// TwinCAT 3 PLC project ExternControl
// ProgramVersion: 3.1.4026.22
// libraries:
//   Tc2_Standard, * (Beckhoff Automation GmbH)
//   Tc2_System, * (Beckhoff Automation GmbH)
//   Tc2_Utilities, * (Beckhoff Automation GmbH)
// project tree:
//   CAM/types/ ST_CAM_CTRL.TcDUT, ST_CAM_DATA.TcDUT (not stored), ST_CAM_INFO.TcDUT (not stored), ST_CAM_OPTIONS.TcDUT (not stored), ST_CAM_READ_VALUES_PARAMETER.TcDUT, ST_CAM_SCALING_DATA.TcDUT, ST_CAM_STATE.TcDUT (not stored), ST_MOTION_FUNCTION.TcDUT, ST_MOTION_FUNCTION_POINT.TcDUT (not stored)
//   FLYING_SAW/ GVL_FLYING_SAW.TcGVL
//   FLYING_SAW/types/ ST_FLY_CTRL.TcDUT (not stored), ST_FLY_DATA.TcDUT (not stored), ST_FLY_OPTIONS.TcDUT (not stored), ST_FLY_STATE.TcDUT (not stored), ST_FLY_SYNC_MODE.TcDUT (not stored)
//   FUNCTIONS/TOUCH_PROBE/types/ ST_2BIT.TcDUT (not stored), ST_CTRL_TOUCH_PROBE.TcDUT, ST_DC_Input.TcDUT, ST_MTI_INPUT.TcDUT, ST_MTI_STATUS.TcDUT, ST_STATE_TOUCH_PROBE.TcDUT
//   FUNCTIONS/TRIGGER_BOX/types/ ST_CTRL_TRIGGER.TcDUT, ST_DC_Output.TcDUT (not stored), ST_DC_State.TcDUT (not stored), ST_STATE_TRIGGER.TcDUT (not stored), T_TriggerControlBits.TcDUT (not stored)
//   / GlobalTextList.TcGTLO (not stored), MAIN.TcPOU, PlcTask.TcTTO, Visualization Manager.TcVMO (not stored)
//   MAPPING/ MAPPING_out.TcPOU, MAPPING_in.TcPOU
//   MAPPING/types/ U_AXIS_CTRL.TcDUT (not stored), U_AXIS_GEAR_IN.TcDUT (not stored), U_AXIS_HOMING.TcDUT (not stored), U_AXIS_INFO.TcDUT (not stored), U_AXIS_MOTION_OPTIONS.TcDUT, U_AXIS_MOVE_DATA.TcDUT (not stored), U_AXIS_NC_PARAMETER_RD.TcDUT, U_AXIS_NC_PARAMETER_WRT.TcDUT (not stored), U_AXIS_STATE.TcDUT (not stored), U_CAM_CTRL.TcDUT (not stored), U_CAM_DATA.TcDUT (not stored), U_CAM_INFO.TcDUT, U_CAM_STATE.TcDUT (not stored), U_FLY_CTRL.TcDUT, U_FLY_DATA.TcDUT, U_FLY_OPTIONS.TcDUT, U_FLY_STATE.TcDUT, U_NCI_AXIS_ID_GROUP.TcDUT (not stored), U_NCI_CTRL.TcDUT (not stored), U_NCI_INDEX_GROUP.TcDUT, U_NCI_R_PARAMETER_I.TcDUT, U_NCI_R_PARAMETER_Q.TcDUT, U_NCI_STATE.TcDUT, U_TOUCH_PROBE_CTRL.TcDUT, U_TOUCH_PROBE_STATE.TcDUT (not stored), U_TRIGGER_CTRL.TcDUT, U_TRIGGER_STATE.TcDUT (not stored)
//   NCI/types/ E_NCI_CHANNEL_ERROR.TcDUT (not stored), E_NCI_CTRL.TcDUT (not stored), E_NCI_INTERPRETER_STATE.TcDUT, E_NCI_STATE.TcDUT (not stored), ST_3D_Group.TcDUT, ST_Index_Group.TcDUT (not stored), ST_Interface_Group.TcDUT (not stored), ST_NciChannel_Ref.TcDUT, ST_NCI_CTRL.TcDUT, ST_NCI_M_FUNC.TcDUT, ST_NCI_STATE.TcDUT (not stored), ST_R_Parameter.TcDUT
//   NC_PTP/types/axis/ E_AxisEncoderType.TcDUT, ST_HomeParams.TcDUT (not stored), ST_HomingOptionsExt.TcDUT
//   NC_PTP/types/control/ E_AXIS_CTRL.TcDUT (not stored), E_AXIS_STATE.TcDUT (not stored), ST_AXIS_CTRL.TcDUT, ST_AXIS_INFO.TcDUT (not stored), ST_AXIS_STATE.TcDUT (not stored), ST_GEAR_IN.TcDUT, ST_HOMING.TcDUT (not stored), ST_MOTION_OPTIONS.TcDUT (not stored), ST_MOVE_DATA.TcDUT, ST_NC_PARAMETER.TcDUT (not stored)
//   TEST_MOTION/ TEST.TcPOU
//   _DUT/ f_GetProgress.TcPOU, f_GetState.TcPOU, E_CHECK_STATE.TcDUT, E_PROGRESS.TcDUT
//   _GVL/ GVL_AXIS.TcGVL, GVL_CAM.TcGVL (not stored), GVL_FUNCTIONS.TcGVL (not stored), GVL_MSG.TcGVL, PLC_CONSTANT.TcGVL
//   _MSG/ fb_LocalTime.TcPOU, fb_MessageData.TcPOU, fb_MessageDataCtrl.TcPOU, f_MessageSet.TcPOU, I_MessageData.TcIO
//   _MSG/types/ e_Device.TcDUT, E_MessageType.TcDUT, E_MESSAGE_BATCH.TcDUT, E_MESSAGE_CHECK.TcDUT, E_MESSAGE_CTRL.TcDUT, E_MESSAGE_FLOW.TcDUT, E_MESSAGE_STATE.TcDUT, e_Subdevice.TcDUT, ST_Message.TcDUT, ST_MESSAGE_CTRL.TcDUT, ST_MESSAGE_STATE.TcDUT, TL_E_MESSAGETYPE.TcTLO
// real-time tasks:
//   TASK PlcTask: cycle T#1ms, priority 20, ADS port 350
//   TASK PlcTask1: cycle T#1ms, priority 1, ADS port 351
// motion (NC):
//   TASK NC-Task 1 SAF: cycle T#2ms, priority 4, ADS port 501
//   TASK NC-Task 1 SVB: cycle T#10ms, priority 8, ADS port 511
//   AXIS Axis 1 (id 1)
//     OtherSettings: AllowMotionCmdToSlave=true
//     encoder EncType=1
//     drive DrvType=5
//       Analog: TorqueSetpointScale=10, ScaleFactorActTorque=0.1
//       TimeComp: TaskDelayCycles=1
//     controller CtrType=1
//       CtrPara: PriorControlFactor=1
//         Observer: BandWidth=20
//   AXIS Axis 2 (id 2)
//     OtherSettings: AllowMotionCmdToSlave=true
//     encoder EncType=1
//     drive DrvType=5
//       Analog: TorqueSetpointScale=10, ScaleFactorActTorque=0.1
//       TimeComp: TaskDelayCycles=1
//     controller CtrType=1
//       CtrPara: PriorControlFactor=1
//         Observer: BandWidth=20
//   AXIS Axis 3 (id 3)
//     OtherSettings: AllowMotionCmdToSlave=true
//     encoder EncType=1
//     drive DrvType=5
//       Analog: TorqueSetpointScale=10, ScaleFactorActTorque=0.1
//       TimeComp: TaskDelayCycles=1
//     controller CtrType=1
//       CtrPara: PriorControlFactor=1
//         Observer: BandWidth=20
//   AXIS Axis 4 (id 4)
//     OtherSettings: AllowMotionCmdToSlave=true
//     encoder EncType=1
//     drive DrvType=5
//       Analog: TorqueSetpointScale=10, ScaleFactorActTorque=0.1
//       TimeComp: TaskDelayCycles=1
//     controller CtrType=1
//       CtrPara: PriorControlFactor=1
//         Observer: BandWidth=20
//   AXIS Axis 5 (id 5)
//     OtherSettings: AllowMotionCmdToSlave=true
//     encoder EncType=1
//     drive DrvType=5
//       Analog: TorqueSetpointScale=10, ScaleFactorActTorque=0.1
//       TimeComp: TaskDelayCycles=1
//     controller CtrType=1
//       CtrPara: PriorControlFactor=1
//         Observer: BandWidth=20
//   AXIS Axis 6 (id 6)
//     OtherSettings: AllowMotionCmdToSlave=true
//     encoder EncType=1
//     drive DrvType=5
//       Analog: TorqueSetpointScale=10, ScaleFactorActTorque=0.1
//       TimeComp: TaskDelayCycles=1
//     controller CtrType=1
//       CtrPara: PriorControlFactor=1
//         Observer: BandWidth=20
// variable links:
//   ExternControl/ExternControl Instance <-> PLC_MOTION/PLC_MOTION Instance
//     PlcTask Inputs/MAIN.eInitPlcMotion <-> PlcTask Outputs/MAIN_AXIS.eInit
//     PlcTask Inputs/MAPPING_in.AxisInfo.byState <-> PlcTask Outputs/MAPPING_AXIS_out.AxisInfo.byState
//     PlcTask Inputs/MAPPING_in.AxisParameterRd.byState <-> PlcTask Outputs/MAPPING_AXIS_out.AxisParameterOut.byState
//     PlcTask Inputs/MAPPING_in.AxisState.byState <-> PlcTask Outputs/MAPPING_AXIS_out.AxisState.byState
//     PlcTask Inputs/MAPPING_in.FlyState.byState <-> PlcTask Outputs/MAPPING_AXIS_out.FlyState.byState
//     PlcTask Outputs/MAPPING_out.AxisCtrl.byCtrl <-> PlcTask Inputs/MAPPING_AXIS_in.AxisCtrl.byCtrl
//     PlcTask Outputs/MAPPING_out.AxisGearInData.byCtrl <-> PlcTask Inputs/MAPPING_AXIS_in.AxisGearInData.byCtrl
//     PlcTask Outputs/MAPPING_out.AxisHoming.byCtrl <-> PlcTask Inputs/MAPPING_AXIS_in.AxisHoming.byCtrl
//     PlcTask Outputs/MAPPING_out.AxisMotionOptions.byCtrl <-> PlcTask Inputs/MAPPING_AXIS_in.AxisMotionOptions.byCtrl
//     PlcTask Outputs/MAPPING_out.AxisMoveData.byCtrl <-> PlcTask Inputs/MAPPING_AXIS_in.AxisMoveData.byCtrl
//     PlcTask Outputs/MAPPING_out.AxisParameterWrt.byCtrl <-> PlcTask Inputs/MAPPING_AXIS_in.AxisParameterIn.byCtrl
//     PlcTask Outputs/MAPPING_out.FlyControl.byCtrl <-> PlcTask Inputs/MAPPING_AXIS_in.FlyControl.byCtrl
//     PlcTask Outputs/MAPPING_out.FlyData.byCtrl <-> PlcTask Inputs/MAPPING_AXIS_in.FlyData.byCtrl
//     PlcTask Outputs/MAPPING_out.FlyOptions.byCtrl <-> PlcTask Inputs/MAPPING_AXIS_in.FlyOptions.byCtrl
//   PLC_MOTION/PLC_MOTION Instance <-> NC-Task 1 SAF/Axes/Axis 1
//     PlcTask Inputs/GVL_AXIS.AxisRef[1].NcToPlc <-> Outputs/ToPlc
//     PlcTask Outputs/GVL_AXIS.AxisRef[1].PlcToNc <-> Inputs/FromPlc
//   PLC_MOTION/PLC_MOTION Instance <-> NC-Task 1 SAF/Axes/Axis 2
//     PlcTask Inputs/GVL_AXIS.AxisRef[2].NcToPlc <-> Outputs/ToPlc
//     PlcTask Outputs/GVL_AXIS.AxisRef[2].PlcToNc <-> Inputs/FromPlc
//   PLC_MOTION/PLC_MOTION Instance <-> NC-Task 1 SAF/Axes/Axis 3
//     PlcTask Inputs/GVL_AXIS.AxisRef[3].NcToPlc <-> Outputs/ToPlc
//     PlcTask Outputs/GVL_AXIS.AxisRef[3].PlcToNc <-> Inputs/FromPlc
//   PLC_MOTION/PLC_MOTION Instance <-> NC-Task 1 SAF/Axes/Axis 4
//     PlcTask Inputs/GVL_AXIS.AxisRef[4].NcToPlc <-> Outputs/ToPlc
//     PlcTask Outputs/GVL_AXIS.AxisRef[4].PlcToNc <-> Inputs/FromPlc
//   PLC_MOTION/PLC_MOTION Instance <-> NC-Task 1 SAF/Axes/Axis 5
//     PlcTask Inputs/GVL_AXIS.AxisRef[5].NcToPlc <-> Outputs/ToPlc
//     PlcTask Outputs/GVL_AXIS.AxisRef[5].PlcToNc <-> Inputs/FromPlc
//   PLC_MOTION/PLC_MOTION Instance <-> NC-Task 1 SAF/Axes/Axis 6
//     PlcTask Inputs/GVL_AXIS.AxisRef[6].NcToPlc <-> Outputs/ToPlc
//     PlcTask Outputs/GVL_AXIS.AxisRef[6].PlcToNc <-> Inputs/FromPlc

CONFIGURATION ExternControl
    RESOURCE PLC ON TwinCAT3
        TASK PlcTask(INTERVAL := T#1ms, PRIORITY := 20);
        PROGRAM MAPPING_in WITH PlcTask : MAPPING_in;
        PROGRAM MAIN WITH PlcTask : MAIN;
        PROGRAM MAPPING_out WITH PlcTask : MAPPING_out;
    END_RESOURCE
END_CONFIGURATION

// ---- CAM/types/ST_CAM_CTRL.TcDUT
{attribute 'pack_mode' := '2'}
TYPE ST_CAM_CTRL :
STRUCT
  eCmd               : E_AXIS_CTRL;    // commanded axis function
END_STRUCT
END_TYPE

// ---- CAM/types/ST_CAM_READ_VALUES_PARAMETER.TcDUT
{attribute 'pack_mode' := '2'}
TYPE ST_CAM_READ_VALUES_PARAMETER :
STRUCT
  nValueSelectMask        : UINT;   // ReadMotionFunctionValues
  rValueMasterStart       : LREAL;  // ReadMotionFunctionValues
  rValueMasterEnd         : LREAL;  // ReadMotionFunctionValues
  rIncrement              : LREAL;
END_STRUCT
END_TYPE

// ---- CAM/types/ST_CAM_SCALING_DATA.TcDUT
{attribute 'pack_mode' := '2'}
TYPE ST_CAM_SCALING_DATA :
STRUCT
  bMasterRelative         : BIT;
  bSlaveRelative          : BIT;

  // scaling of X-axis (Master) of the CAM
  nMasterScalingMode      : UINT;
  rMasterOffset           : LREAL;
  rMasterScaling          : LREAL := 1.0;

  // scaling of Y-axis (Slave) of CAM
  nSlaveScalingMode       : UINT;

  rSlaveOffset            : LREAL;
  rSlaveScaling           : LREAL := 1.0;
END_STRUCT
END_TYPE

// ---- CAM/types/ST_MOTION_FUNCTION.TcDUT
{attribute 'pack_mode' := '2'}
TYPE ST_MOTION_FUNCTION :
STRUCT
  stMotionFunction            : ARRAY[1..MAX_MOTION_FUNCTION_POINTS] OF ST_MOTION_FUNCTION_POINT;
  nMotionFunctionSize         : UINT;
  nPoints                     : UINT; // number of points used in motion function 
END_STRUCT
END_TYPE

// ---- FUNCTIONS/TOUCH_PROBE/types/ST_CTRL_TOUCH_PROBE.TcDUT
TYPE ST_CTRL_TOUCH_PROBE :
STRUCT
  Enable        : BIT;

  AxisId        : UDINT;      // TwinCAT NC Axis ID

  SensorIndex   : UDINT;      // sensor select; 1 := upper , 2 := lower, 0 := default upper 

  Direction     : INT := 1;   // typeof(MC_DIRECTION)
                                // MC_Positive_Direction := 1,   -(set trigger when crossing moving in pos dir)
                                // MC_Shortest_Way,               (not used in TouchProbe or TriggerBox)
                                // MC_Negative_Direction := 3,   -(set trigger when crossing moving in neg dir)
                                // MC_Current_Direction  := 4,    (not used in TouchProbe or TriggerBox)
                                // MC_Undefined_Direction := 128  (not used in TouchProbe or TriggerBox)

  PositionStart : LREAL; // axis has to reach this position in order to start the check for change in input timestamp
  PositionEnd   : LREAL; // axis must not reach this position without state change on input --> error
END_STRUCT
END_TYPE

// ---- FUNCTIONS/TOUCH_PROBE/types/ST_DC_Input.TcDUT
TYPE ST_DC_Input :
STRUCT
  Input      : BIT;

  Status     : USINT;

  LatchPositive  : ULINT;
  LatchNegative  : ULINT;
END_STRUCT
END_TYPE

// ---- FUNCTIONS/TOUCH_PROBE/types/ST_MTI_INPUT.TcDUT
TYPE ST_MTI_INPUT :
STRUCT
  EventState            : BIT;
  EventTime             : UDINT;
END_STRUCT
END_TYPE

// ---- FUNCTIONS/TOUCH_PROBE/types/ST_MTI_STATUS.TcDUT
TYPE ST_MTI_STATUS :
STRUCT
  EventCount            : USINT;
  InputState            : BIT;
  InputBufferOverflow   : BIT;
  InputCycleCounter     : ST_2BIT;
  CountsInBuffer        : USINT;
  InputOrderFeedback    : usint;
END_STRUCT
END_TYPE

// ---- FUNCTIONS/TOUCH_PROBE/types/ST_STATE_TOUCH_PROBE.TcDUT
TYPE ST_STATE_TOUCH_PROBE :
STRUCT
  State           : UINT;   // 0 := deactivated, 100 := BUSY, 1000 := DONE, 9000 := ERROR
  LatchPositive   : LREAL;  // rising edge
  LatchNegative   : LREAL;  // falling edge
END_STRUCT
END_TYPE

// ---- FUNCTIONS/TRIGGER_BOX/types/ST_CTRL_TRIGGER.TcDUT
TYPE ST_CTRL_TRIGGER :
STRUCT
  Control             : T_TriggerControlBits;

   {attribute 'hide'}
  byc : ARRAY[1..7] OF BYTE;;


  AxisId              : UDINT;  // TwinCAT NC Axis ID

  TriggerCount        : UDINT;  // how many TriggerPositions shall be used

  TriggerPosition     : ARRAY[1..MAX_TRIGGER_COUNT] OF LREAL;  // Axis Position where output must be set by TriggerBox
                                // Trigger is set when crossing Position
END_STRUCT
END_TYPE

// ---- MAPPING/types/U_AXIS_MOTION_OPTIONS.TcDUT
TYPE U_AXIS_MOTION_OPTIONS :
UNION

  stCtrl              : ARRAY[1..MAX_AXIS] OF ST_MOTION_OPTIONS;

  byCtrl    AT %Q*    : ARRAY[1..MAX_AXIS] OF
                        ARRAY[1..SIZEOF(ST_MOTION_OPTIONS)] OF BYTE;
END_UNION
END_TYPE

// ---- MAPPING/types/U_AXIS_NC_PARAMETER_RD.TcDUT
TYPE U_AXIS_NC_PARAMETER_RD :
UNION

  stState             : ARRAY[1..MAX_AXIS] OF ST_NC_PARAMETER;

  byState   AT %I*    : ARRAY[1..MAX_AXIS] OF
                        ARRAY[1..SIZEOF(ST_NC_PARAMETER)] OF BYTE;
END_UNION
END_TYPE

// ---- MAPPING/types/U_CAM_INFO.TcDUT
TYPE U_CAM_INFO :
UNION

  stState             : ARRAY[1..MAX_AXIS] OF ST_CAM_INFO;

  byState  AT %i*     : ARRAY[1..MAX_AXIS] OF
                        ARRAY[1..SIZEOF(ST_CAM_INFO)] OF BYTE;
END_UNION
END_TYPE

// ---- MAPPING/types/U_FLY_CTRL.TcDUT
TYPE U_FLY_CTRL :
UNION

  stCtrl              : ARRAY[1..MAX_AXIS] OF ST_FLY_CTRL;

  byCtrl    AT %Q*    : ARRAY[1..MAX_AXIS] OF
                        ARRAY[1..SIZEOF(ST_FLY_CTRL)] OF BYTE;

END_UNION
END_TYPE

// ---- MAPPING/types/U_FLY_DATA.TcDUT
TYPE U_FLY_DATA :
UNION

  stCtrl              : ARRAY[1..MAX_AXIS] OF ST_FLY_DATA;

  byCtrl    AT %Q*    : ARRAY[1..MAX_AXIS] OF
                        ARRAY[1..SIZEOF(ST_FLY_DATA)] OF BYTE;

END_UNION
END_TYPE

// ---- MAPPING/types/U_FLY_OPTIONS.TcDUT
TYPE U_FLY_OPTIONS :
UNION

  stCtrl              : ARRAY[1..MAX_AXIS] OF ST_FLY_OPTIONS;

  byCtrl    AT %Q*    : ARRAY[1..MAX_AXIS] OF
                        ARRAY[1..SIZEOF(ST_FLY_OPTIONS)] OF BYTE;

END_UNION
END_TYPE

// ---- MAPPING/types/U_FLY_STATE.TcDUT
TYPE U_FLY_STATE :
UNION

  stState             : ARRAY[1..MAX_AXIS] OF ST_FLY_STATE;

  byState   AT %I*    : ARRAY[1..MAX_AXIS] OF
                        ARRAY[1..SIZEOF(ST_FLY_STATE)] OF BYTE;
END_UNION
END_TYPE

// ---- MAPPING/types/U_NCI_INDEX_GROUP.TcDUT
TYPE U_NCI_INDEX_GROUP :
UNION

  stCtrl              : ARRAY[1..MAX_NCI_CH] OF ST_Index_Group;

  byCtrl    AT %q*    : ARRAY[1..MAX_NCI_CH] OF
                        ARRAY[1..SIZEOF(ST_Index_Group)] OF BYTE;
END_UNION
END_TYPE

// ---- MAPPING/types/U_NCI_R_PARAMETER_I.TcDUT
TYPE U_NCI_R_PARAMETER_I :
UNION

  stCtrl              : ARRAY[1..MAX_NCI_CH] OF ST_R_Parameter;

  byCtrl    AT %q*    : ARRAY[1..MAX_NCI_CH] OF
                        ARRAY[1..SIZEOF(ST_R_Parameter)] OF BYTE;
END_UNION
END_TYPE

// ---- MAPPING/types/U_NCI_R_PARAMETER_Q.TcDUT
TYPE U_NCI_R_PARAMETER_Q :
UNION

  stCtrl              : ARRAY[1..MAX_NCI_CH] OF ST_R_Parameter;

  byCtrl    AT %i*    : ARRAY[1..MAX_NCI_CH] OF
                        ARRAY[1..SIZEOF(ST_R_Parameter)] OF BYTE;
END_UNION
END_TYPE

// ---- MAPPING/types/U_NCI_STATE.TcDUT
TYPE U_NCI_STATE :
UNION

  stState             : ARRAY[1..MAX_NCI_CH] OF ST_NCI_STATE;

  byState   AT %i*    : ARRAY[1..MAX_NCI_CH] OF
                        ARRAY[1..SIZEOF(ST_NCI_STATE)] OF BYTE;
END_UNION
END_TYPE

// ---- MAPPING/types/U_TOUCH_PROBE_CTRL.TcDUT
TYPE U_TOUCH_PROBE_CTRL :
UNION
  stCtrl              : ARRAY[1..MAX_TOUCH_PROBE] OF ST_CTRL_TOUCH_PROBE;

  byCtrl    AT %q*    : ARRAY[1..MAX_TOUCH_PROBE] OF
                        ARRAY[1..SIZEOF(ST_CTRL_TOUCH_PROBE)] OF BYTE;
END_UNION
END_TYPE

// ---- MAPPING/types/U_TRIGGER_CTRL.TcDUT
TYPE U_TRIGGER_CTRL :
UNION
  stCtrl              : ARRAY[1..MAX_TRIGGER_BOX] OF ST_CTRL_TRIGGER;

  byCtrl    AT %q*    : ARRAY[1..MAX_TRIGGER_BOX] OF
                        ARRAY[1..SIZEOF(ST_CTRL_TRIGGER)] OF BYTE;
END_UNION
END_TYPE

// ---- NCI/types/E_NCI_INTERPRETER_STATE.TcDUT
// Interpreter state, see also library tc2_nci.Global_Variables.NCI_INTERPRETER_xxx
//  Date    Name  Version   Remarks
//  2016/09/29  FJK   1.0     1st Version
{attribute -'to_string'}
TYPE E_NCI_INTERPRETER_STATE :
(
  NCI_INTERPRETER_INITFAILED := 0,
  NCI_INTERPRETER_IDLE := 1,
  NCI_INTERPRETER_READY := 2,
  NCI_INTERPRETER_STARTED := 3,
  NCI_INTERPRETER_SCANNING := 4,
  NCI_INTERPRETER_RUNNING := 5,
  NCI_INTERPRETER_STAY_RUNNING := 6,
  NCI_INTERPRETER_WRITETABLE := 7,
  NCI_INTERPRETER_SEARCHLINE := 8,
  NCI_INTERPRETER_END := 9,
  NCI_INTERPRETER_SINGLESTOP := 10, 
  NCI_INTERPRETER_ABORTING := 11,
  NCI_INTERPRETER_ABORTED := 12,
  NCI_INTERPRETER_FAULT := 13,
  NCI_INTERPRETER_RESET := 14,
  NCI_INTERPRETER_STOP := 15,
  NCI_INTERPRETER_WAITFUNC := 16,
  NCI_INTERPRETER_FLUSHBUFFERS := 17
) DWORD;    //Basis-Datentyp
END_TYPE

// ---- NCI/types/ST_3D_Group.TcDUT
{attribute 'pack_mode' := '2'}
TYPE ST_3D_Group :
STRUCT
  nXAxisId    : UDINT := 1;
  nYAxisId    : UDINT := 2;
  nZAxisId    : UDINT := 3;
  nQ1AxisId   : UDINT;
  nQ2AxisId   : UDINT;
  nQ3AxisId   : UDINT;
  nQ4AxisId   : UDINT;
  nQ5AxisId   : UDINT;
END_STRUCT
END_TYPE

// ---- NCI/types/ST_NciChannel_Ref.TcDUT
TYPE ST_NciChannel_Ref :
STRUCT
  NcToPlc AT %I*: NcToPlc_NciChannel_Ref;   //  Externer Datentyp!
  PlcToNc AT %Q*: PlcToNc_NciChannel_Ref;   //  Externer Datentyp!
END_STRUCT
END_TYPE

// ---- NCI/types/ST_NCI_CTRL.TcDUT
{attribute 'pack_mode' := '2'}
TYPE ST_NCI_CTRL :
STRUCT
  eCmd          : E_NCI_CTRL := E_NCI_CTRL.INIT;
  rOverride     : REAL := 47.11;

  sProgramName  : STRING(255);
END_STRUCT
END_TYPE

// ---- NCI/types/ST_NCI_M_FUNC.TcDUT
{attribute 'pack_mode' := '2'}
TYPE ST_NCI_M_FUNC :
STRUCT
  FastMFuncMask   : ARRAY [1..5] OF DWORD;
  HskMFuncNo      : UINT;
  HskMFuncReq     : WORD;
  HFuncValue      : UDINT; 

  MFuncGranted    : UINT;
END_STRUCT
END_TYPE

// ---- NCI/types/ST_R_Parameter.TcDUT
{attribute 'pack_mode' := '2'}
TYPE ST_R_Parameter :
STRUCT
  _nStart               : DINT := 901;
  _nCount               : DINT :=   4;
  _rValue               : ARRAY[0..MAX_R_PARA] OF LREAL;
END_STRUCT
END_TYPE

// ---- NC_PTP/types/axis/E_AxisEncoderType.TcDUT
{attribute 'to_string'}
TYPE E_AxisEncoderType :
(
  NoEncoder := 0,
  
  Simulation_Encoder,
  
  M3000_Enc,
  M31x0_M2000_Enc,
  MDP_511_Enc,
  MDP_500_501_Enc,
  MDP_510_Enc,
  KL30xx_Enc,
  SERCOS_EtherCAT_SoE_Pos,
  SERCOS_EtherCAT_SoE_Pos_Velo,
  Binary_Enc,
  M2510_Enc,
  FOX50_Enc                     := 12,
  AX2000_Lightbus               := 14,
  Provi_DriveMC_Simodrive_611U,
  Universal_Encoder_varBitmask,
  NC_Backplane,
  spec_CANopen_Typ,
  MDP_513_DS402,
  AX2xx_B900,
  KL5151_Encoder                := 21,
  IP5209_Encoder                := 24,
  KL2531_KL2541_Encoder,
  KL2532_KL2542_Encoder,
  Time_Base_Encoder,
  TCom_Encoder_SoftDrive
)UDINT;
END_TYPE

// ---- NC_PTP/types/axis/ST_HomingOptionsExt.TcDUT
TYPE ST_HomingOptionsExt :
STRUCT
  // in order for extern control to be 
  // fully independent of any library types
  // struct is built with base types
  ClearPositionLag      : BOOL;
  SearchDirection       : INT;    // MC_Direction
  SearchVelocity        : LREAL;
  SyncDirection         : INT;    // MC_Direction
  SyncVelocity          : LREAL;
  ReferenceMode         : UDINT;  // E_EncoderReferenceMode
END_STRUCT
END_TYPE

// ---- NC_PTP/types/control/ST_AXIS_CTRL.TcDUT
{attribute 'pack_mode' := '2'}
TYPE ST_AXIS_CTRL :
STRUCT
  eCmd                : E_AXIS_CTRL;    // commanded axis function
  eProgress           : E_PROGRESS;     // progress command for synced functions
END_STRUCT
END_TYPE

// ---- NC_PTP/types/control/ST_GEAR_IN.TcDUT
{attribute 'pack_mode' := '2'}
TYPE ST_GEAR_IN :
STRUCT
  bAdvancedSlaveDynamics  : BOOL;
  nMultiMasterSyncMode    : INT;

  nAxisIndexMaster    : ARRAY [1..4] OF BYTE; // Index of Master1-4
  rGearRatio          : ARRAY [1..4] OF REAL; 
  Acceleration        : REAL;
  Deceleration        : REAL;
  Jerk                : REAL;  
END_STRUCT
END_TYPE

// ---- NC_PTP/types/control/ST_MOVE_DATA.TcDUT
{attribute 'pack_mode' := '2'}
TYPE ST_MOVE_DATA :
STRUCT
  rSetPos           : LREAL;
  rSetVelo          : LREAL;
  rOverride         : LREAL := 100.0;
  rAcc              : LREAL;
  rDec              : LREAL;
  rJerk             : LREAL;
  iDirection        : INT;
END_STRUCT
END_TYPE

// ---- _DUT/E_CHECK_STATE.TcDUT
{attribute 'qualified_only'}
{attribute 'strict'}
{attribute 'to_string'}
TYPE E_CHECK_STATE :
(
  CHECK_INIT,
  AXIS_INDEX_OUT_OF_RANGE         :=  10,

	AXIS_REF_POINTER_INVALID        := 100,
  AXIS_CTRL_POINTER_INVALID,
  AXIS_STATE_POINTER_INVALID,
  AXIS_INFO_POINTER_INVALID,
  AXIS_DATA_POINTER_INVALID,
  AXIS_NC_PARAMETER_POINTER_INVALID,
  AXIS_HOME_PARAMETER_POINTER_INVALID,
  AXIS_GEAR_IN_PARAMETER_POINTER_INVALID,
  AXIS_GEAR_IN_MULTIMASTER_POINTER_INVALID,
  AXIS_MOTION_OPTIONS_POINTER_INVALID,

  NCI_NOT_ACTIVATED               := 200,
  NCI_CHANNEL_REF_POINTER_INVALID,
  NCI_AXIS_CONFIG_POINTER_INVALID,
  NCI_MCS_AXIS_POINTER_INVALID,
  NCI_AUX_AXIS_POINTER_INVALID,
  NCI_CTRL_POINTER_INVALID,
  NCI_STATE_POINTER_INVALID,
  NCI_R_PARAMETER_READ_POINTER_INVALID,
  NCI_R_PARAMETER_wRITE_POINTER_INVALID,
  NCI_M_FUNC_POINTER_INVALID,

  CAM_NOT_ACTIVATED               := 300,
  CAM_SLAVE_AXIS_REF_INVALID,
  CAM_SLAVE_ITF_MC_AXIS_INVALID,
  CAM_MASTER_AXIS_REF_INVALID,
  CAM_MOTION_FUNCTION_POINTER_INVALID,
  CAM_MOTION_FUNCTION_POINT_POINTER_INVALID,

  CHECK_DONE                      := 10000
  
)UINT;
END_TYPE

// ---- _DUT/E_PROGRESS.TcDUT
{attribute 'qualified_only'}
//{attribute 'strict'}
{attribute 'to_string'}
TYPE E_PROGRESS :
(
  // progress has 2 use cases
  // 1. as offset to cyclic interface's state 
  //    for the requested command/function
  //    e.g. State := <Enum equivalent to eCmd> + E_PROGRESS
  //
  // 2. as state feedback (result) from (any) method
  PROGRESS_INVALID,
  PROGRESS_NOT_EXIST      :=   100,
  PROGRESS_INIT           :=  1000,
  PROGRESS_BUSY           :=  2000,
  PROGRESS_PREPARE        :=  3000,
  PROGRESS_STARTUP        :=  4000,
  PROGRESS_CHECK          :=  5000,
  PROGRESS_OCCUPIED       :=  6000,
  PROGRESS_WORKING        :=  7000,
  PROGRESS_STILL_WORKING  :=  8000,
  PROGRESS_ERROR          :=  9000,
  PROGRESS_DONE           := 10000
)UINT;
END_TYPE

// ---- _MSG/types/e_Device.TcDUT
{attribute 'to_string'}
TYPE e_Device :
(
  // txt file logging LOG_FILE
  Device_Null,                // NULL           - not to be used
  Device_Main,                // MAIN(PRG)      - reserved for MAIN(PRG)
  Device_Nci,                 // NCI(PRG)       - reserved for NCI(PRG)
  Device_Cam,                 // CAM(PRG        - reserved for CAM(PRG)
  Device_Functions,           // FUNCTIONS(PRG) - reserved for FUNCTIONS(PRG)

  General           :=  1000,
  CaGroup           :=  2000,
  Xpu               :=  3000,
  XpuCtrl           :=  4000,
  Mover             :=  5000,
  MoverCtrl         :=  6000,
  XtsTransportUnit  :=  7000,
  XfcTriggerBox     :=  8000,
  XfcTouchProbe     :=  9000,
  XtsStation        := 10000,

  Camming           := 11000,
  NciChannel        := 12000,
  NciChannelCtrl    := 13000,
  Axis              := 14000,
  XfcAxis           := 15000,

  // txt file logging LOG_FILE_METRICS
  Metrics           := 16000,

  // txt file logging LOG_FILE_APP
  Process           := 20000,
  ProcessListCtrl   := 21000,
  TicketListCtrl    := 22000,

  Application       := 30000,

  // txt file logging LOG_FILE_PRODUCT - this is for you to use
  DataProduct       := 40000
)UDINT;
END_TYPE

// ---- _MSG/types/E_MessageType.TcDUT
{attribute 'strict'}
{attribute 'to_string'}
TYPE E_MessageType :
(
  //-----------------------------------------------------
  //-----------------------------------------------------
  //  message system:
  //  - errors are always calling f_MessageSet()
  //  - errors are always entered into its list
  //
  //  - message severity is set by this enum (like everywhere else)
  //
  //  - message frequency is set by this enum
  //    - IF you get above 50 stations, 
  //      writing to the file system takes time:
  //
  //    Batch: switching on metrics (> Empty) must not add cpu load, 
  //      --> so do not clutter here
  //
  //    Info:  regular flow of information (>Error / >Warning) 
  //           must not add significant cpu load, 
  //      --> so do not clutter here
  //
  //    Verbose and above:
  //    --> for small systems (< 96 mover, < 50 stations) 
  //        you may switch it on for everybody, 
  //        files get big quickly ;-)
  //
  //    --> switch on during test phase for a handful of stations
  //
  //    --> high detail logging always and for everybody
  //    --> we need somebody who transfers data more quickly
  //      --> I can offer a .NET(C#) ADS tool which collects the list.
  //          .NET application then pushes to database
  //-----------------------------------------------------
  //-----------------------------------------------------
  eMessageEmpty,    // he who is without bounds may speak
  eMessageBatch,    // he who counts words, counts numbers (Batch started, Next in Batch, Batch done)
  eMessageError,    // mine, your(')s, anybody's, let the numbers tell you
  eMessageWarning,  // I told you so
  eMessageInfo,     // A long time ago in a galaxy far, far away...
  eMessageVerbose,  // He talks a lot, doesn't he?; Yeah! He's very knowledgeable.
  eMessageSentient  // Keep them out of bright light, Don't get them wet, do not feed them after midnight!! No matter how much they beg!!
)DINT;
END_TYPE

// ---- _MSG/types/E_MESSAGE_BATCH.TcDUT
{attribute 'qualified_only'}
{attribute 'strict'}
{attribute 'to_string'}
TYPE E_MESSAGE_BATCH :
(
	MSG_BATCH_NULL,
  MSG_BATCH_JOB_STARTED,
  MSG_BATCH_NEXT_IN_JOB,
  MSG_BATCH_JOB_DONE
)UINT;
END_TYPE

// ---- _MSG/types/E_MESSAGE_CHECK.TcDUT
{attribute 'qualified_only'}
{attribute 'strict'}
{attribute 'to_string'}
TYPE E_MESSAGE_CHECK :
(
  // 9000 --> here comes your error
  MSG_CHECK_INVALID_POINTER             := 9000,
  MSG_CHECK_INVALID_POINTER_TIME,
  MSG_CHECK_INVALID_POINTER_LIST,
  MSG_CHECK_INVALID_POINTER_MSG_IDX,
  MSG_CHECK_INVALID_POINTER_ERR_IDX,
  MSG_CHECK_INVALID_POINTER_ROOT_FILE,
  MSG_CHECK_INVALID_POINTER_ROOT_DIR,
  MSG_CHECK_INVALID_POINTER_CTRL,
  MSG_CHECK_INVALID_POINTER_STATE,

  // 10000 --> here comes your man
  MSG_CHECK_DONE                        := 10000
)UINT;
END_TYPE

// ---- _MSG/types/E_MESSAGE_CTRL.TcDUT
{attribute 'qualified_only'}
{attribute 'strict'}
{attribute 'to_string'}
TYPE E_MESSAGE_CTRL :
(
	MSG_CTRL_NULL,
	MSG_CTRL_INIT   := 10,
  MSG_CTRL_IDLE   := 30,
  MSG_CTRL_WRITE  := 50
)UINT;
END_TYPE

// ---- _MSG/types/E_MESSAGE_FLOW.TcDUT
{attribute 'qualified_only'}
{attribute 'strict'}
{attribute 'to_string'}
TYPE E_MESSAGE_FLOW :
(
  MSG_FLOW_INIT,
  MSG_FLOW_ROOT                 := 10,
  MSG_FLOW_ROOT_CREATE,
  MSG_FLOW_ROOT_CREATE_BUSY,
  MSG_FLOW_FOLDER,
  MSG_FLOW_FOLDER_CREATE,
  MSG_FLOW_FOLDER_CREATE_BUSY,
  MSG_FLOW_FILE_CREATE_DONE,
  MSG_FLOW_LINE_START           := 100,
  MSG_FLOW_LINE_BUILD,
  MSG_FLOW_LINE_CHECK,
  MSG_FLOW_WRITE_FILE_BUSY      := 200,
  MSG_FLOW_WRITE_FILE_END,
  MSG_FLOW_WRITE_FILE_DONE      := 1000
)UINT;
END_TYPE

// ---- _MSG/types/E_MESSAGE_STATE.TcDUT
{attribute 'qualified_only'}
//{attribute 'strict'}
{attribute 'to_string'}
TYPE E_MESSAGE_STATE :
(
	MSG_STATE_NULL,
  MSG_STATE_INIT    := 10,
  MSG_STATE_IDLE    := 30,
  MSG_STATE_WRITE   := 50
)UINT;
END_TYPE

// ---- _MSG/types/e_Subdevice.TcDUT
{attribute 'strict'}
{attribute 'to_string'}
TYPE e_Subdevice :
(
  // sub device for message system
  General                 :=  0,
  MainInit,
  // Motion Control FB Instances
  fbPower,
  fbReset,
  fbResetSercos,
  fbHalt,
  fbStop,                 // 5
  fbHome,
  fbJog,
  fbMoveVelocity1,
  fbMoveVelocity2,
  fbMoveAbsolute1,        // 10
  fbMoveAbsolute2,
  fbMoveEndless,
  fbMovePtP,
  fbMoveVelo,

  // CA CollisionAvoidance FB instances
  // CA group fb instances
  fbCaGroup             := 30,
  fbMoveToPosCa,
  fbSendToAbsPosCa,
  fbSendToModuloPosCa,
  fbGearInPosCa,
  fbGroupAddAxis,
  fbGroupRemoveAxis,
  fbGroupDisable,
  fbGroupEnable,
  fbGroupErrorRead,
  fbGroupStatusRead,
  fbGroupReset,
  fbGroupStop,
  fbHaltCa,
  fbSendToPos,

  fbGearIn                := 50,
  fbGearOut,
  fbGearInMultiMaster,

  fbCamOut                := 80,
  fbCamInV2,
  fbCamScalingV2,
  fbCamInfoV2,
  fbReadMotionFunction,
  fbReadMotionFunctionPoint,
  fbReadMotionFunctionValues,
  fbWriteMotionFunction,
  fbWriteMotionFunctionPoint,
  fbSetOnlineChangeMode,

  fbReadParameter         := 100,
  fbReadBoolParameter,
  fbWriteParameter,
  fbWriteBoolParameter,
  fbWriteParameterPersistent,

  fbBuildGroup            := 200,
  fbClearGroup,
  fbLoadProg,
  fbResetItp,
  fbStartStopItp,
  fbEStopItp,             // 205
  fbStepOnAfterEStopItp,
  fbConfirmHskItp,
  fbDelDtgItp,
  fbNciFeedTablePreparation,
  fbNciFeedTable,         // 210
  fbReadLine,
  fbItpReadRParams,
  fbItpWriteRParams,
  Get_ItpState,
  Get_Error,              // 215


  XfcPositionAtTime       := 300,
  XfcTimeOfPosition,
  XfcTimeToPosition,
  XfcTimeToModuloPosition,
  XfcRecordedPosition,
  XfcTouchProbe,          // 305
  XfcTouchProbeEL1258,
  XfcTouchProbeOptions,
  XfcTriggerRef,
  XfcTriggerRef_MT,
  XfcEl1258Interface_MT,  // 310
  XfcRecordedPosition_MT,
  XfcTriggerOut,
  XfcTriggerStart,
  XfcSwitchOn_2252,
  XfcSwitchOff_2252,      // 315
  XfcInit,
  XfcLatchPosition,
  XfcWaitForPosition,

  AxisMode              := 1000,
  AxisControl,
  AxisStartUp,
  AxisCycle,
  AxisIdle,

  NciControl            := 2000,
  NciStartUp,
  NciCycle,
  NciIdle,

  StationLinkedList     := 3000,
  StationInitList,
  StationAddHead,
  StationAddTail,
  StationGetHead,
  StationRemoveHeadValue,
  StationGearInDistanceToSync,
  StationGearInSyncStart,
  StationGearInSyncMove,
  StationGearInSyncEnd,

  StationControl        := 4000,
  StationState, 

  Xpu_fbEnvironment     := 5000,
  Xpu_fbProcessingUnit,
  Xpu_fbXpuPart,
  Xpu_fbXpuTrack,
  Xpu_fbMc2CaGroup,
  Xpu_fbParameterSet,
  Xpu_fbNctController,

  Xpu_fbPartModules     := 5500,

  Xpu_fbMoverXpu        := 6000,

  Xpu_fbNctBaseUnit     := 6500,

  TransportUnit_General := 7000,
  TransportUnit_Restart := 7010,
  TransportUnit_Start,
  TransportUnit_XpuInit,
  TransportUnit_StationClearOutfeed,

  CamControl            := 8000,
  CamStartUp,
  CamCycle,

  Process_StationCollector    := 11000,
  Process_ProcessCollector    := 11100,
  Process_ProcessCollector_Init,
  Process_ProcessCollector_Cycle,
  Process_ProcessCollector_Control,

  Process_LinkedList_GetHead,
  Process_LinkedList_RemoveHead,
  Process_LinkedList_AddTail,
  Process_LinkedList_CheckData,
  Process_StationQueue_Check,

  Process_LinkedList_Com              := 11200,
  Process_LinkedList_Com_Init,
  Process_LinkedList_Com_Cmd,
  Process_LinkedList_Com_AddHead,
  Process_LinkedList_Com_AddTail,
  Process_LinkedList_Com_DelHead,
  Process_LinkedList_Com_DelTail,
  Process_LinkedList_Com_GetHead,
  Process_LinkedList_Com_GetTail,


  Instance_Command              := 12000,
  Instance_ProcessConductor,
  Instance_BufferInfeed,
  Instance_Infeed,
  Instance_BufferOutfeed,
  Instance_Outfeed,
  Instance_Sender_Buffer,

  Ticket_LinkedList_Ctrl        := 12100,
  Ticket_LinkedList_Com_Init,
  Ticket_LinkedList_Com_Cmd,
  Ticket_LinkedList_Com_AddHead,
  Ticket_LinkedList_Com_AddTail,
  Ticket_LinkedList_Com_DelHead,
  Ticket_LinkedList_Com_DelTail,
  Ticket_LinkedList_Com_GetHead,
  Ticket_LinkedList_Com_GetTail,
  

  Application                 := 13000,
  Application_Check,
  Application_Clear,
  Application_Cmd,
  Application_Disable,
  Application_Enable,
  Application_Finish,
  Application_Init,
  Application_Proceed,
  Application_Work


)DINT;
END_TYPE

// ---- _MSG/types/ST_Message.TcDUT
TYPE ST_Message :
STRUCT
  eType         : e_MessageType;
  eDevice       : e_Device;
  eSubdevice    : e_SubDevice;
  {attribute 'displaymode':='hex'}
  iErrorNumber  : ULINT;
  tTime         : STRING(24);
  sText         : STRING(127);
END_STRUCT
END_TYPE

// ---- _MSG/types/ST_MESSAGE_CTRL.TcDUT
TYPE ST_MESSAGE_CTRL :
STRUCT
  Cmd         : E_MESSAGE_CTRL;
END_STRUCT
END_TYPE

// ---- _MSG/types/ST_MESSAGE_STATE.TcDUT
TYPE ST_MESSAGE_STATE :
STRUCT
  State         : E_MESSAGE_STATE;  // as always... combined value of Cmd equivalent and e_progress
END_STRUCT
END_TYPE

// ---- FLYING_SAW/GVL_FLYING_SAW.TcGVL
{attribute 'qualified_only'}
VAR_GLOBAL
  //-----------------------------------------------------------------------------
  // command and state structure
  //  - datafields for anyone to access
  //    - ADS via symbol
  //    - cyclic mapping to any other cyclic network/runtime
  //-----------------------------------------------------------------------------
  Ctrl                        : ARRAY[1..PLC_CONSTANT.MAX_AXIS] OF ST_FLY_CTRL;      // command structure to write into
  State                       : ARRAY[1..PLC_CONSTANT.MAX_AXIS] OF ST_FLY_STATE;     // state structure to read from


  //-----------------------------------------------------------------------------
  // data and info structure
  //  - parameter data fields for
  //    - Ctrl  --> Data
  //    - State --> Info
  //-----------------------------------------------------------------------------
//  Info                        : ARRAY[1..PLC_CONSTANT.MAX_AXIS] OF ST_FLY_INFO;
  Data                        : ARRAY[1..PLC_CONSTANT.MAX_AXIS] OF ST_FLY_DATA;


  //-----------------------------------------------------------------------------
  // R/W datafields
  // - optional data for CheckMask
  // - The Options contains two position values as limits. 
  //   The check for these position limits can be activated. 
  //   To do this, two flags 
  //   (GearInSync_CheckMask_OptionalMinPos, 
  //    GearInSync_CheckMask_OptionalMaxPos) 
  //   have to be set in the SyncMode structure.
  //
  //-----------------------------------------------------------------------------
  Options                     : ARRAY[1..PLC_CONSTANT.MAX_AXIS] OF ST_FLY_OPTIONS;

END_VAR

// ---- _GVL/GVL_AXIS.TcGVL
{attribute 'qualified_only'}
VAR_GLOBAL
  //-----------------------------------------------------------------------------
  // command and state structure
  //  - datafields for anyone to access
  //    - ADS via symbol
  //    - cyclic mapping to any other cyclic network/runtime
  //-----------------------------------------------------------------------------
  Ctrl                        : ARRAY[1..PLC_CONSTANT.MAX_AXIS] OF ST_AXIS_CTRL;      // command structure to write into
  State                       : ARRAY[1..PLC_CONSTANT.MAX_AXIS] OF ST_AXIS_STATE;     // state structure to read from

  //-----------------------------------------------------------------------------
  // data and info structure
  //  - parameter data fields for
  //    - Ctrl  --> Data
  //    - State --> Info
  //-----------------------------------------------------------------------------
  Info                        : ARRAY[1..PLC_CONSTANT.MAX_AXIS] OF ST_AXIS_INFO;      // axis state and position data to read from
  Data                        : ARRAY[1..PLC_CONSTANT.MAX_AXIS] OF ST_MOVE_DATA;      // axis data to write into


  //-----------------------------------------------------------------------------
  // special function parameter structs
  // - additional details for axis command
  //-----------------------------------------------------------------------------
  NcParameterWrt              : ARRAY[1..PLC_CONSTANT.MAX_AXIS] OF ST_NC_PARAMETER;   // struct for a single parameter value put/get your data here before/after using Ctrl
  NcParameterRd               : ARRAY[1..PLC_CONSTANT.MAX_AXIS] OF ST_NC_PARAMETER;   // struct for a single parameter value put/get your data here before/after using Ctrl

  HomeParameter               : ARRAY[1..PLC_CONSTANT.MAX_AXIS] OF ST_HOMING;         // homing parameter for each axis

  GearInParameter             : ARRAY[1..PLC_CONSTANT.MAX_AXIS] OF ST_GEAR_IN;        // GearIn and GearInMultiMaster, index to master axes[1-4], rGearRatio[1-4]

  MotionOptions               : ARRAY[1..PLC_CONSTANT.MAX_AXIS] OF ST_MOTION_OPTIONS; // additional motion parameters
END_VAR

// ---- _GVL/GVL_MSG.TcGVL
{attribute 'qualified_only'}
VAR_GLOBAL CONSTANT
  //-----------------------------------------------------------------------------
  // file paths for message system
  //  - compiler define option WIN switches to Windows file paths
  //-----------------------------------------------------------------------------
{IF NOT defined (BSD)}
  {info 'EXT_MOTION_CONTROL: WIN'}
  LOG_DIR               : STRING  := 'C:\TwinCAT\#MsgFiles\';
{ELSE}
  {info 'EXT_MOTION_CONTROL: BSD'}
  LOG_DIR               : STRING  := '/usr/local/etc/TwinCAT/#MsgFiles/';
{END_IF}

  LOG_FILE              : STRING  := concat(TO_STRING(TwinCAT_SystemInfoVarList._AppInfo.AdsPort), '_MSG_PLC_');
  LOG_FILE_METRIC       : STRING  := concat(TO_STRING(TwinCAT_SystemInfoVarList._AppInfo.AdsPort), '_MSG_Metrics_');

  MAX_MESSAGE           : UINT    := 200; // max entry in message list
END_VAR
VAR_GLOBAL
  //-----------------------------------------------------------------------------
  // Message System
  //  - Everybody uses f_MessageSet(ST_Message)
  //    - DECISION WHICH LIST IS MADE IN f_MessageSet !!
  //    - which list to use is determined by e_Device in your message
  //
  //  - MessageData instances are self sufficient and need only 
  //    datafield assignment for correct data-flow
  //
  //
  //-----------------------------------------------------------------------------
  //-----------------------------------------------------------------------------
  //-----------------------------------------------------------------------------
  // (ST_Message.eDevice := from Device_Null to XfcAxis)
  //-----------------------------------------------------------------------------
  MotionMessageData               : fb_MessageDataCtrl;
  MotionMessageCtrl               : st_message_ctrl;
  MotionMessageState              : st_message_state;

  MotionMessages                  : ARRAY[1..MAX_MESSAGE] OF ST_Message;
  MessageMotionIndex              : UINT := 0; // message index for base layer
  MessageMotionError              : UINT := 0; // error counter for base layer
  //-----------------------------------------------------------------------------
  //-----------------------------------------------------------------------------
  // (ST_Message.eDevice := e_Device.Metrics)
  //-----------------------------------------------------------------------------
  MetricMessageData               : fb_MessageDataCtrl;
  MetricMessageCtrl               : st_message_ctrl;
  MetricMessageState              : st_message_state;

  MetricMessages                  : ARRAY[1..MAX_MESSAGE] OF ST_Message;
  MessageMetricIndex              : UINT := 0; // message index for metrics data
  MessageMetricError              : UINT := 0; // error counter for metrics data
  //-----------------------------------------------------------------------------
  //-----------------------------------------------------------------------------
  fbLocalTime                     : fb_LocalTime;
  dtLocalTime                     : DT;
  sLocalTime                      : STRING;
  //-----------------------------------------------------------------------------
  //-----------------------------------------------------------------------------
  //-----------------------------------------------------------------------------
  //-----------------------------------------------------------------------------
{IF defined (TEST)}
  {info 'TEST logging enabled'}
  MessageLevel                    : E_MessageType := eMessageverbose; // a lot of messages
{ELSE}
  MessageLevel                    : E_MessageType := eMessageEmpty; // only errors are written into list 
{END_IF}

  MessageLevelAxisPtp             : ARRAY[1..PLC_CONSTANT.MAX_AXIS]   OF E_MessageType;
  MessageLevelAxisCam             : ARRAY[1..PLC_CONSTANT.MAX_AXIS]   OF E_MessageType;
  MessageLevelNciChn              : ARRAY[1..PLC_CONSTANT.MAX_NCI_CH] OF E_MessageType;

  MessageLevelTriggerBox          : ARRAY[1..PLC_CONSTANT.MAX_TRIGGER_BOX]  OF E_MessageType;
  MessageLevelTouchProbe          : ARRAY[1..PLC_CONSTANT.MAX_TOUCH_PROBE]  OF E_MessageType;

END_VAR

// ---- _GVL/PLC_CONSTANT.TcGVL
//{attribute 'qualified_only'}
VAR_GLOBAL CONSTANT


  //-----------------------------------------------------------------------------
  // AXIS related limits
  //-----------------------------------------------------------------------------
  MAX_AXIS              : UINT    := 6;
  MAX_RETRY             : UINT    := 5;


  //-----------------------------------------------------------------------------
  // NCI related limits and *.nc standard folder
  //-----------------------------------------------------------------------------
{IF NOT defined (BSD)}
  NCI_DIR               : STRING  := 'C:\TwinCAT\Mc\Nci\';
{ELSE}
  NCI_DIR               : STRING  := '/usr/local/etc/TwinCAT/Mc/Nci/';
{END_IF}

{IF defined (NCI)}
  {info 'PLC_MOTION_LAYER: NCI'}
  NCI_ACTIVE            : BOOL    := TRUE;
  CONFIG_NAME           : STRING  := 'NCI_Spec_Ch_';
{ELSE}
  NCI_ACTIVE            : BOOL    := FALSE;
  CONFIG_NAME           : STRING  := 'NCI_NOT_ACTIVE';
{END_IF}

  MAX_NCI_CH            : UINT    := 1;

  MAX_PATH_STEPS        : UINT    := 5;
  MAX_MC_AXIS           : UINT    := 3;
  MAX_AUX_AXIS          : UINT    := 2;
  MAX_R_PARA            : UINT    := 10;


  //-----------------------------------------------------------------------------
  // CAMMING related limits
  //-----------------------------------------------------------------------------
{IF defined (CAM)}
  {info 'PLC_MOTION_LAYER: CAM'}
  CAM_ACTIVE                  : BOOL    := TRUE;
{ELSE}
  CAM_ACTIVE                  : BOOL    := FALSE;
{END_IF}

  MAX_CAM_CH                  : UINT    := 1;

  MAX_MOTION_FUNCTION_POINTS  : UINT    := 10;

  // HAUD
  // 17.07.2024
  // Start Implementation of Position Trigger function
  //  - Timestamp/position output
  //  - Latch DC time from input
  
  MAX_TRIGGER_BOX   : UINT := 12;
  MAX_TOUCH_PROBE   : UINT := 12;

  MAX_TRIGGER_COUNT : UINT :=  4;

  MAX_MTI_CH        : UINT :=  1; // MAX mti channel per EL terminal

{IF defined (XFC)}
  {info 'PLC_MOTION_LAYER: XFC'}
  XFC_ACTIVE        : BOOL := TRUE;
{ELSE}
  XFC_ACTIVE        : BOOL := FALSE;
{END_IF}

END_VAR

// ---- _MSG/I_MessageData.TcIO
INTERFACE I_MessageData

PROPERTY DirRoot : POINTER to string(255)
SET
END_SET
END_PROPERTY

PROPERTY ErrorIndex : reference to uint
SET
END_SET
END_PROPERTY

PROPERTY FileRoot : pointer to string(255)
SET
END_SET
END_PROPERTY

PROPERTY LocalTime : pointer to DT
SET
END_SET
END_PROPERTY

PROPERTY MessageIndex : reference to uint
SET
END_SET
END_PROPERTY

PROPERTY MsgList : pointer to ARRAY[1..GVL_MSG.MAX_MESSAGE] OF st_message
SET
END_SET
END_PROPERTY

END_INTERFACE

// ---- MAPPING/MAPPING_in.TcPOU
PROGRAM MAPPING_in
VAR
  bFirstCycle           : BOOL := TRUE;

  AxisState             : U_AXIS_STATE;
  AxisInfo              : U_AXIS_INFO;
  AxisParameterRd       : U_AXIS_NC_PARAMETER_RD;

  CamState              : U_CAM_STATE;
  CamInfo               : U_CAM_INFO;

  TriggerState          : U_TRIGGER_STATE;

  TouchState            : U_TOUCH_PROBE_STATE;

  FlyState              : U_FLY_STATE;


  szAxisPara,
  szAxisInfo,
  szAxisState           : ARRAY[1..2] OF UDINT;

  szCamInfo,
  szCamData,
  szCamState            : ARRAY[1..2] OF UDINT;

  szStateTouchProbe,
  szStateTrigger	      :  ARRAY[1..2] OF UDINT;
END_VAR


IF (bFirstCycle)
THEN
  bFirstCycle         := FALSE;
  
  szAxisState[1]      := SIZEOF(AxisState);
  szAxisState[2]      := SIZEOF(GVL_AXIS.State);
  
  szAxisInfo [1]      := SIZEOF(AxisInfo);
  szAxisInfo [2]      := SIZEOF(GVL_AXIS.Info);
  
  szAxisPara [1]      := SIZEOF(AxisParameterRd);
  szAxisPara [2]      := SIZEOF(GVL_AXIS.NcParameterRd);
END_IF

  memcpy(ADR(GVL_AXIS.State),             ADR(AxisState),              SIZEOF(AxisState));
  memcpy(ADR(GVL_AXIS.Info),              ADR(AxisInfo),               SIZEOF(AxisInfo));
  memcpy(ADR(GVL_AXIS.NcParameterRd),     ADR(AxisParameterRd),        SIZEOF(AxisParameterRd));

  memcpy(ADR(GVL_CAM.State),              ADR(CamState),               SIZEOF(CamState));
  memcpy(ADR(GVL_CAM.Info),               ADR(CamInfo),                SIZEOF(CamInfo));

  memcpy(ADR(GVL_FUNCTIONS.StateTrigger),    ADR(TriggerState),        SIZEOF(TriggerState));
  memcpy(ADR(GVL_FUNCTIONS.StateTouchProbe), ADR(TouchState),          SIZEOF(TouchState));

  memcpy(ADR(GVL_FLYING_SAW.State),       ADR(FlyState),               SIZEOF(FlyState));

END_PROGRAM

// ---- MAIN.TcPOU
//-----------------------------------------------------------------------------------------------------------------
// ExternControl: EXT_MOTION_CONTROL
//
// BASIC EXAMPLE for controlling PLC_MOTION_LAYER
//-----------------------------------------------------------------------------------------------------------------
PROGRAM MAIN
VAR
  //---------------------------------------------------------------------------------------------------------------
  eInitPlcMotion  AT %I*  : E_PROGRESS;   // startup indicator from PLC_MOTION plc
  //---------------------------------------------------------------------------------------------------------------

  nAxis           : UINT := 1;  // you choose

  bStartAxis,
  bStartCam       : BOOL;

  eStateAxis,
  eStateCam       : E_PROGRESS;

  eCtrlFunction   : E_AXIS_CTRL   := E_AXIS_CTRL.AXIS_ENABLE;   // for you to set
  eStateFunction  : E_AXIS_STATE  := E_AXIS_STATE.AXIS_ENABLE;  // for you to set so the result can be checked correctly

  stMsg           : ST_Message;
  eMsgState       : e_message_state;
  eMsgProgress    : E_PROGRESS;
END_VAR

//-----------------------------------------------------------------------------------------------------------------
// Local time; used for timestamps
//-----------------------------------------------------------------------------------------------------------------
GVL_MSG.fbLocalTime(
                    sLocalTime                => GVL_MSG.sLocalTime, 
                    dtLocalTime               => GVL_MSG.dtLocalTime);
//-----------------------------------------------------------------------------------------------------------------
//-----------------------------------------------------------------------------------------------------------------
// PLC_MOTION_LAYER startup check: 
//  - you may evaluate this on your own terms
//  - putting it here was convenient for me in the context of this simple example
//-----------------------------------------------------------------------------------------------------------------
//-----------------------------------------------------------------------------------------------------------------
IF NOT (eInitPlcMotion = E_PROGRESS.PROGRESS_DONE)
THEN
  RETURN;
END_IF
//-----------------------------------------------------------------------------------------------------------------
//-----------------------------------------------------------------------------------------------------------------
// BASIC SEQUENCE for controlling PLC_MOTION_LAYER
//-----------------------------------------------------------------------------------------------------------------
//-----------------------------------------------------------------------------------------------------------------
TEST();
//-----------------------------------------------------------------------------------------------------------------
//-----------------------------------------------------------------------------------------------------------------
// BASIC EXAMPLE for controlling PLC_MOTION_LAYER
//-----------------------------------------------------------------------------------------------------------------
//-----------------------------------------------------------------------------------------------------------------
//-----------------------------------------------------------------------------------------------------------------
// HOW to... PtP axis
//  - you have to use the data and parameter fields in the matching GVL
//-----------------------------------------------------------------------------------------------------------------
IF NOT bStartAxis
THEN
  // this is for cleaning up your state machine
  eStateAxis                      := E_PROGRESS.PROGRESS_INIT;
END_IF
//-----------------------------------------------------------------------------------------------------------------
//-----------------------------------------------------------------------------------------------------------------
CASE eStateAxis 
OF
  E_PROGRESS.PROGRESS_INIT:
    IF bStartAxis                 // do not forget to set the motion data for the chosen axis, GVL_AXIS.Data etc. 
    THEN
      GVL_AXIS.Ctrl[nAxis].eCmd   := eCtrlFunction;

      eStateAxis                  := E_PROGRESS.PROGRESS_BUSY;
    END_IF


  E_PROGRESS.PROGRESS_BUSY:
    IF (GVL_AXIS.State[nAxis].eState = eStateFunction + E_PROGRESS.PROGRESS_DONE)
    THEN
      eStateAxis                  := E_PROGRESS.PROGRESS_DONE;

    ELSIF (GVL_AXIS.State[nAxis].eState = eStateFunction + E_PROGRESS.PROGRESS_ERROR)
    THEN
      eStateAxis                  := E_PROGRESS.PROGRESS_ERROR;
    END_IF
END_CASE
//-----------------------------------------------------------------------------------------------------------------
//-----------------------------------------------------------------------------------------------------------------
// HOW to... CAM axis
//  - you have to use the data and parameter fields in the matching GVL
//-----------------------------------------------------------------------------------------------------------------
IF NOT bStartCam
THEN
  // this is for cleaning up your state machine
  eStateCam                       := E_PROGRESS.PROGRESS_INIT;
END_IF
//-----------------------------------------------------------------------------------------------------------------
//-----------------------------------------------------------------------------------------------------------------
CASE eStateCam
OF
  E_PROGRESS.PROGRESS_INIT:
    IF bStartCam                 // do not forget to set the motion data for the chosen axis, GVL_AXIS.Data etc. 
    THEN
      GVL_CAM.Ctrl[nAxis].eCmd    := eCtrlFunction;

      eStateCam                   := E_PROGRESS.PROGRESS_BUSY;
    END_IF


  E_PROGRESS.PROGRESS_BUSY:
    IF (GVL_AXIS.State[nAxis].eState = eStateFunction + E_PROGRESS.PROGRESS_DONE)
    THEN
      eStateCam                   := E_PROGRESS.PROGRESS_DONE;

    ELSIF (GVL_AXIS.State[nAxis].eState = eStateFunction + E_PROGRESS.PROGRESS_ERROR)
    THEN
      eStateCam                   := E_PROGRESS.PROGRESS_ERROR;
    END_IF
END_CASE
//-----------------------------------------------------------------------------------------------------------------
//-----------------------------------------------------------------------------------------------------------------
//-----------------------------------------------------------------------------------------------------------------
//  /logging
//    - all life is problem solving
//-----------------------------------------------------------------------------------------------------------------
GVL_MSG.MotionMessageData.Ctrl                REF= GVL_MSG.MotionMessageCtrl;
GVL_MSG.MotionMessageData.State               REF= GVL_MSG.MotionMessageState;

GVL_MSG.MotionMessageData.MessageIndex        REF= GVL_MSG.MessageMotionIndex;
GVL_MSG.MotionMessageData.ErrorIndex          REF= GVL_MSG.MessageMotionError;

GVL_MSG.MotionMessageData.DirRoot             :=   ADR(GVL_MSG.LOG_DIR);
GVL_MSG.MotionMessageData.FileRoot            :=   ADR(GVL_MSG.LOG_FILE);

GVL_MSG.MotionMessageData.MsgList             :=   ADR(GVL_MSG.MotionMessages);
GVL_MSG.MotionMessageData.LocalTime           :=   ADR(GVL_MSG.dtLocalTime);

GVL_MSG.MotionMessageData();               

eMsgState                                     :=   f_GetState   (GVL_MSG.MotionMessageState.State);
eMsgProgress                                  :=   f_GetProgress(GVL_MSG.MotionMessageState.State);

CASE eMsgState
OF
  E_MESSAGE_STATE.MSG_STATE_NULL:
    CASE eMsgProgress
    OF
      E_PROGRESS.PROGRESS_INVALID,
      E_PROGRESS.PROGRESS_DONE:
        IF (GVL_MSG.MessageMotionIndex > GVL_MSG.MAX_MESSAGE/100) OR
           (GVL_MSG.MessageMotionError > 0)
        THEN
          GVL_MSG.MotionMessageCtrl.Cmd       := E_MESSAGE_CTRL.MSG_CTRL_WRITE;
        END_IF
    END_CASE

  E_MESSAGE_STATE.MSG_STATE_WRITE:
    CASE eMsgProgress
    OF
      E_PROGRESS.PROGRESS_ERROR,
      E_PROGRESS.PROGRESS_DONE:
        GVL_MSG.MotionMessageCtrl.Cmd         := E_MESSAGE_CTRL.MSG_CTRL_NULL;
    END_CASE

ELSE
    CASE eMsgProgress
    OF
      E_PROGRESS.PROGRESS_DONE:
        GVL_MSG.MotionMessageCtrl.Cmd         := E_MESSAGE_CTRL.MSG_CTRL_NULL;
    END_CASE
END_CASE
//-----------------------------------------------------------------------------------------------------------------
//  logging/
//-----------------------------------------------------------------------------------------------------------------
//-----------------------------------------------------------------------------------------------------------------

END_PROGRAM

// ---- TEST_MOTION/TEST.TcPOU
//-----------------------------------------------------------------------------------------------------------------
// ExternControl: EXT_MOTION_CONTROL
//
// BASIC SEQUENCES for controlling PLC_MOTION_LAYER
//  - rudimentary error handling only
//-----------------------------------------------------------------------------------------------------------------
PROGRAM TEST
VAR
  bStart        : BOOL;
  nState,
  nStateNext    : UINT;

  nModulo       : UINT := 10_000;

  nCount,
  nCycle,
  nWait         : UINT;
END_VAR

//-----------------------------------------------------------------------------------------------------------------
//-----------------------------------------------------------------------------------------------------------------
// examples to illustrate Ctrl/State use
//-----------------------------------------------------------------------------------------------------------------
//-----------------------------------------------------------------------------------------------------------------
CASE nState
OF
  0,
  10:
    IF bStart
    THEN
      nCount                    :=   0;
      nCycle                    :=   5;
      nState                    := 100;
    END_IF


  100:
    GVL_AXIS.Ctrl[1].eCmd       := E_AXIS_CTRL.AXIS_ENABLE;
    IF (GVL_AXIS.State[1].eState = E_AXIS_STATE.AXIS_ENABLE + E_PROGRESS.PROGRESS_ERROR)
    THEN
      nState                    := 9000;  // error reaction required, e.g. RESET

    ELSIF (GVL_AXIS.State[1].eState = E_AXIS_STATE.AXIS_ENABLE + E_PROGRESS.PROGRESS_DONE)
    THEN
      nState                    := 101;
    END_IF

  101:
    GVL_AXIS.Ctrl[2].eCmd       := E_AXIS_CTRL.AXIS_ENABLE;
    IF (GVL_AXIS.State[2].eState = E_AXIS_STATE.AXIS_ENABLE + E_PROGRESS.PROGRESS_ERROR)
    THEN
      nState                    := 9001;  // error reaction required, e.g. RESET

    ELSIF (GVL_AXIS.State[2].eState = E_AXIS_STATE.AXIS_ENABLE + E_PROGRESS.PROGRESS_DONE)
    THEN
      nState                    := 102;
    END_IF

  102:
    GVL_AXIS.Ctrl[3].eCmd       := E_AXIS_CTRL.AXIS_ENABLE;
    IF (GVL_AXIS.State[3].eState = E_AXIS_STATE.AXIS_ENABLE + E_PROGRESS.PROGRESS_ERROR)
    THEN
      nState                    := 9002;  // error reaction required, e.g. RESET

    ELSIF (GVL_AXIS.State[3].eState = E_AXIS_STATE.AXIS_ENABLE + E_PROGRESS.PROGRESS_DONE)
    THEN
      nState                    := 110;
    END_IF

  110:
    GVL_AXIS.Data[1].rSetPos    :=   3141.59;
    GVL_AXIS.Data[1].rSetVelo   :=    271.82;
    GVL_AXIS.Data[1].rAcc       :=   9810.00;
    GVL_AXIS.Data[1].rDec       :=   9810.00;
    GVL_AXIS.Data[1].rJerk      := 299792.46;

    GVL_AXIS.Ctrl[1].eCmd       := E_AXIS_CTRL.AXIS_MOVE_POS;
    IF (GVL_AXIS.State[1].eState = E_AXIS_STATE.AXIS_MOVE_POS + E_PROGRESS.PROGRESS_ERROR)
    THEN
      nState                    := 9010;  // error reaction required, e.g. RESET

    ELSIF (GVL_AXIS.State[1].eState = E_AXIS_STATE.AXIS_MOVE_POS + E_PROGRESS.PROGRESS_DONE)
    THEN
      GVL_AXIS.Ctrl[1].eCmd     := E_AXIS_CTRL.AXIS_NULL;
      nState                    := 120;
    END_IF

  120:
    GVL_AXIS.Data[2].rSetVelo   :=    666.00;
    GVL_AXIS.Data[2].rAcc       :=  15000.00;
    GVL_AXIS.Data[2].rDec       :=  15000.00;
    GVL_AXIS.Data[2].rJerk      := 300000.00;
    GVL_AXIS.Data[2].iDirection :=      1;

    GVL_AXIS.Ctrl[2].eCmd       := E_AXIS_CTRL.AXIS_MOVE_VELO;
    IF (GVL_AXIS.State[2].eState = E_AXIS_STATE.AXIS_MOVE_VELO + E_PROGRESS.PROGRESS_ERROR)
    THEN
      nState                    := 9020;  // error reaction required, e.g. RESET

    ELSIF (GVL_AXIS.State[2].eState = E_AXIS_STATE.AXIS_MOVE_VELO + E_PROGRESS.PROGRESS_DONE)
    THEN
      nState                    := 1000;
      nStateNext                :=  125;
    END_IF

  125:
    GVL_AXIS.Data[1].rSetPos    :=   2718.28;
    GVL_AXIS.Data[1].rSetVelo   :=    314.15;
    GVL_AXIS.Data[1].rAcc       :=   9810.00;
    GVL_AXIS.Data[1].rDec       :=   9810.00;
    GVL_AXIS.Data[1].rJerk      := 299792.46;

    GVL_AXIS.Ctrl[1].eCmd       := E_AXIS_CTRL.AXIS_MOVE_POS;
    IF (GVL_AXIS.State[1].eState = E_AXIS_STATE.AXIS_MOVE_POS + E_PROGRESS.PROGRESS_ERROR)
    THEN
      nState                    := 9010;  // error reaction required, e.g. RESET

    ELSIF (GVL_AXIS.State[1].eState = E_AXIS_STATE.AXIS_MOVE_POS + E_PROGRESS.PROGRESS_DONE)
    THEN
      nState                    := 130;
    END_IF


  130:
    GVL_AXIS.Data[3].rSetVelo   :=    707.00;
    GVL_AXIS.Data[3].rAcc       :=  15000.00;
    GVL_AXIS.Data[3].rDec       :=  15000.00;
    GVL_AXIS.Data[3].rJerk      := 300000.00;
    GVL_AXIS.Data[3].iDirection :=     -1;

    GVL_AXIS.Ctrl[3].eCmd       := E_AXIS_CTRL.AXIS_MOVE_BUFFER_VELO;
    IF (GVL_AXIS.State[3].eState = E_AXIS_STATE.AXIS_MOVE_BUFFER_VELO + E_PROGRESS.PROGRESS_ERROR)
    THEN
      nState                    := 9300;  // error reaction required, e.g. RESET

    ELSIF (GVL_AXIS.State[3].eState = E_AXIS_STATE.AXIS_MOVE_BUFFER_VELO + E_PROGRESS.PROGRESS_WORKING)
    THEN
      nState                    := 1000;
      nStateNext                :=  140;
    END_IF

  140:
    GVL_AXIS.Data[3].rSetVelo   :=   1414.00;
    GVL_AXIS.Data[3].rAcc       :=  15000.00;
    GVL_AXIS.Data[3].rDec       :=  15000.00;
    GVL_AXIS.Data[3].rJerk      := 300000.00;
    GVL_AXIS.Data[3].iDirection :=     -1;

    GVL_AXIS.Ctrl[3].eCmd       := E_AXIS_CTRL.AXIS_MOVE_BUFFER_VELO;
    IF (GVL_AXIS.State[3].eState = E_AXIS_STATE.AXIS_MOVE_BUFFER_VELO + E_PROGRESS.PROGRESS_ERROR)
    THEN
      nState                    := 9301;  // error reaction required, e.g. RESET

    ELSIF (GVL_AXIS.State[3].eState = E_AXIS_STATE.AXIS_MOVE_BUFFER_VELO + E_PROGRESS.PROGRESS_WORKING)
    THEN
      nState                    := 1000;
      nStateNext                :=  130;
      nCount                    := nCount + 1;
    END_IF

  200:
    GVL_AXIS.Data[3].rSetVelo   :=      0.00;
    GVL_AXIS.Data[3].rAcc       :=  15000.00;
    GVL_AXIS.Data[3].rDec       :=  15000.00;
    GVL_AXIS.Data[3].rJerk      := 300000.00;

    GVL_AXIS.Ctrl[3].eCmd       := E_AXIS_CTRL.AXIS_HALT;
    IF (GVL_AXIS.State[3].eState = E_AXIS_STATE.AXIS_HALT + E_PROGRESS.PROGRESS_ERROR)
    THEN
      nState                    := 9400;  // error reaction required, e.g. RESET

    ELSIF (GVL_AXIS.State[3].eState = E_AXIS_STATE.AXIS_HALT + E_PROGRESS.PROGRESS_DONE)
    THEN
      nState                    :=  201;
    END_IF

  201:
    GVL_AXIS.Data[2].rSetVelo   :=      0.00;
    GVL_AXIS.Data[2].rAcc       :=  15000.00;
    GVL_AXIS.Data[2].rDec       :=  15000.00;
    GVL_AXIS.Data[2].rJerk      := 300000.00;

    GVL_AXIS.Ctrl[2].eCmd       := E_AXIS_CTRL.AXIS_HALT;
    IF (GVL_AXIS.State[2].eState = E_AXIS_STATE.AXIS_HALT + E_PROGRESS.PROGRESS_ERROR)
    THEN
      nState                    := 9500;  // error reaction required, e.g. RESET

    ELSIF (GVL_AXIS.State[2].eState = E_AXIS_STATE.AXIS_HALT + E_PROGRESS.PROGRESS_DONE)
    THEN
      nState                    := 10000;
    END_IF


  1000:
    nWait                       := nWait + 1;
    IF (nWait MOD nModulo = 0)
    THEN
      nWait                     := 1;
      nState                    := nStateNext;

      IF (nCount > nCycle-1)
      THEN
        nState                  := 200;
      END_IF
    END_IF

  10000:
    IF bStart
    THEN
      nState                    := 10; // repeat
    END_IF
END_CASE

END_PROGRAM

// ---- _DUT/f_GetState.TcPOU
// global function to extract state identifier from combined value
FUNCTION f_GetState : uint
VAR_INPUT
  state     : UINT; // combined value of identifier + e_progress
END_VAR
VAR
  _stx      : uint;
END_VAR

_stx          := state MOD E_PROGRESS.PROGRESS_INIT;

IF (_stx = 0)
THEN
  f_GetState  := state;
ELSE
  f_GetState  := _stx;
END_IF

END_FUNCTION

// ---- _DUT/f_GetProgress.TcPOU
// global function to extract e_progress from combined value
FUNCTION f_GetProgress : uint
VAR_INPUT
  state     : UINT;
END_VAR
VAR
  nP        : uint;
END_VAR


nP := state / E_PROGRESS.PROGRESS_INIT;

f_GetProgress := nP * E_PROGRESS.PROGRESS_INIT;

END_FUNCTION

// ---- MAPPING/MAPPING_out.TcPOU
PROGRAM MAPPING_out
VAR
  bFirstCycle       : BOOL := TRUE;

  AxisCtrl          : U_AXIS_CTRL;
  AxisMoveData      : U_AXIS_MOVE_DATA;
  AxisMotionOptions : U_AXIS_MOTION_OPTIONS;

  AxisGearInData    : U_AXIS_GEAR_IN;
  AxisHoming        : U_AXIS_HOMING;
  AxisParameterWrt  : U_AXIS_NC_PARAMETER_WRT;

  CamCtrl           : U_CAM_CTRL;
  CamData           : U_CAM_DATA;

  TriggerCtrl       : U_TRIGGER_CTRL;

  TouchCtrl         : U_TOUCH_PROBE_CTRL;

  FlyControl        : U_FLY_CTRL;
  FlyData           : U_FLY_DATA;
  FlyOptions        : U_FLY_OPTIONS;


  szAxisPara,
  szAxisHoming,
  szAxisGearData,
  szAxisMotionOptions,
  szAxisMoveData,
  szAxisCtrl          : ARRAY[1..2] OF UDINT;

  szCamCtrl           : ARRAY[1..2] OF UDINT;

  szCtrlTouchProbe,
  szCtrlTrigger       :  ARRAY[1..2] OF UDINT;
END_VAR


IF (bFirstCycle)
THEN
  bFirstCycle             := FALSE;

  szAxisCtrl[1]           := SIZEOF(AxisCtrl);
  szAxisCtrl[2]           := SIZEOF(GVL_AXIS.Ctrl);
  
  szAxisMoveData [1]      := SIZEOF(AxisMoveData);
  szAxisMoveData [2]      := SIZEOF(GVL_AXIS.Data);
  
  szAxisMotionOptions [1] := SIZEOF(AxisMotionOptions);
  szAxisMotionOptions [2] := SIZEOF(GVL_AXIS.MotionOptions);
  
  szAxisGearData [1]      := SIZEOF(AxisGearInData);
  szAxisGearData [2]      := SIZEOF(GVL_AXIS.GearInParameter);
  
  szAxisHoming [1]        := SIZEOF(AxisHoming);
  szAxisHoming [2]        := SIZEOF(GVL_AXIS.HomeParameter);
  
  szAxisPara [1]          := SIZEOF(AxisParameterWrt);
  szAxisPara [2]          := SIZEOF(GVL_AXIS.NcParameterWrt);
  
END_IF

  memcpy(ADR(AxisCtrl),                 ADR(GVL_AXIS.Ctrl),             SIZEOF(AxisCTrl));
  memcpy(ADR(AxisMoveData),             ADR(GVL_AXIS.Data),             SIZEOF(AxisMoveData));
  memcpy(ADR(AxisMotionOptions),        ADR(GVL_AXIS.MotionOptions),    SIZEOF(AxisMotionOptions));
  
  memcpy(ADR(AxisGearInData),           ADR(GVL_AXIS.GearInParameter),  SIZEOF(AxisGearInData));
  memcpy(ADR(AxisHoming),               ADR(GVL_AXIS.HomeParameter),    SIZEOF(AxisHoming));
  memcpy(ADR(AxisParameterWrt),         ADR(GVL_AXIS.NcParameterWrt),   SIZEOF(AxisParameterWrt));

  memcpy(ADR(CamCtrl),                  ADR(GVL_CAM.Ctrl),              SIZEOF(CamCtrl));
  memcpy(ADR(CamData),                  ADR(GVL_CAM.Data),              SIZEOF(CamData));

  memcpy(ADR(FlyControl),               ADR(GVL_FLYING_SAW.Ctrl),       SIZEOF(FlyControl));
  memcpy(ADR(FlyData),                  ADR(GVL_FLYING_SAW.Data),       SIZEOF(FlyData));
  memcpy(ADR(FlyOptions),               ADR(GVL_FLYING_SAW.Options),    SIZEOF(FlyOptions));

END_PROGRAM

// ---- _MSG/f_MessageSet.TcPOU
FUNCTION f_MessageSet : BOOL
VAR_INPUT
  stMessage     : ST_Message;
END_VAR
VAR
  _uiIndex      : UINT;
  _MainDevice   : e_Device;
  _nModRes      : UDINT;     // residual after modulo
END_VAR

stMessage.tTime                     := GVL_MSG.sLocalTime;

// why here? so all calls to this function may stay the same
_nModRes                            := stMessage.eDevice MOD e_Device.General;
_MainDevice                         := stMessage.eDevice - _nModRes;

CASE _MainDevice
OF
  (*
  e_device.DataProduct:
    // this is your data, if you choose to use this message system
    FOR _uiIndex := 1 TO GVL_MSG.MAX_MESSAGE
    DO
      IF (GVL_MSG.ProductMessages[_uiIndex].eType = e_MessageType.eMessageEmpty)
      THEN
        GVL_MSG.ProductMessages[_uiIndex]      := stMessage;
        GVL_MSG.MessageProductIndex            := _uiIndex;
        EXIT;
      END_IF
    END_FOR
  
    IF (stMessage.eType = E_MessageType.eMessageError)
    THEN
      // in case of error: increment counter
      GVL_MSG.MessageProductError     := GVL_MSG.MessageProductError + 1;
    END_IF


  e_Device.Process,
  e_Device.Application:
    FOR _uiIndex := 1 TO GVL_MSG.MAX_MESSAGE
    DO
      IF (GVL_MSG.ApplicationMessages[_uiIndex].eType = e_MessageType.eMessageEmpty)
      THEN
        GVL_MSG.ApplicationMessages[_uiIndex]  := stMessage;    // yes, we grab global values directly, only here
        GVL_MSG.MessageApplicationIndex        := _uiIndex;
        EXIT;
      END_IF
    END_FOR
    IF (stMessage.eType = E_MessageType.eMessageError)
    THEN
      // in case of error: increment counter
      GVL_MSG.MessageApplicationError := GVL_MSG.MessageApplicationError + 1;
    END_IF
  *)

  e_Device.Metrics:
    FOR _uiIndex := 1 TO GVL_MSG.MAX_MESSAGE
    DO
      IF (GVL_MSG.MetricMessages[_uiIndex].eType = e_MessageType.eMessageEmpty)
      THEN
        GVL_MSG.MetricMessages[_uiIndex]  := stMessage;    // yes, we grab global values directly, only here
        GVL_MSG.MessageMetricIndex        := _uiIndex;
        EXIT;
      END_IF
    END_FOR
    IF (stMessage.eType = E_MessageType.eMessageError)
    THEN
      // in case of error: increment counter
      GVL_MSG.MessageMetricError := GVL_MSG.MessageMetricError + 1;
    END_IF

ELSE
  FOR _uiIndex := 1 TO GVL_MSG.MAX_MESSAGE
  DO
    IF (GVL_MSG.MotionMessages[_uiIndex].eType = e_MessageType.eMessageEmpty)
    THEN
      GVL_MSG.MotionMessages[_uiIndex]      := stMessage;
      GVL_MSG.MessageMotionIndex            := _uiIndex;
      EXIT;
    END_IF
  END_FOR

  IF (stMessage.eType = E_MessageType.eMessageError)
  THEN
    // in case of error: increment counter
    GVL_MSG.MessageMotionError := GVL_MSG.MessageMotionError + 1;
  END_IF
END_CASE

END_FUNCTION

// ---- _MSG/fb_MessageDataCtrl.TcPOU
FUNCTION_BLOCK fb_MessageDataCtrl EXTENDS fb_MessageData
VAR
  _stCtrl       : REFERENCE TO ST_MESSAGE_CTRL;
  _stState      : REFERENCE TO ST_MESSAGE_STATE;

  _eCmd,
  _eCmdOld      : E_MESSAGE_CTRL;

  _eResult,
  _eJobResult   : E_PROGRESS;

  _eState       : E_MESSAGE_STATE;

END_VAR

//-----------------------------------------------------------------------------
// check pointers
//-----------------------------------------------------------------------------
IF NOT Check()
THEN
  _eResult                      := E_PROGRESS.PROGRESS_ERROR;
  RETURN;
END_IF
//-----------------------------------------------------------------------------
// check date
// new message file for a new day
//-----------------------------------------------------------------------------
IF (FolderDate(_dtLocalTime) <> _sFolderDate)
THEN
  _bFileCreated                 := FALSE;
END_IF
//-----------------------------------------------------------------------------
//----------------------------------------------------------------------------- 
// copy to local for debug
_eCmd                         := _stCtrl.Cmd;

// cyclic check for command change
// get state for cmd
IF (_eCmd <> _eCmdOld)
THEN
  // get matching sdtate for Ctrl.Cmd
  _eState                     := Cmd(_eCmd);
  _eCmdOld                    := _eCmd;
END_IF


CASE _eResult
OF
  E_PROGRESS.PROGRESS_INVALID:
    _stState.State            := E_MESSAGE_STATE.MSG_STATE_NULL;

  E_PROGRESS.PROGRESS_ERROR:
    _stState.State            := _eState + E_PROGRESS.PROGRESS_ERROR;

  E_PROGRESS.PROGRESS_DONE:
    _stState.State            := _eState + E_PROGRESS.PROGRESS_DONE;

ELSE
  // work in progress
  // update progress for extern use
  _stState.State              := _eState + _eResult;

  CASE _eState
  OF
    E_MESSAGE_STATE.MSG_STATE_INIT:
      _eResult                := BuildFolder(TRUE);


    E_MESSAGE_STATE.MSG_STATE_IDLE:
      IF (_nMsgIndex < GVL_MSG.MAX_MESSAGE - GVL_MSG.MAX_MESSAGE/10)
      THEN
        _eResult              := E_PROGRESS.PROGRESS_WORKING;
      ELSE
        _eResult              := E_PROGRESS.PROGRESS_DONE;
        _nMsgIndex            := 0;
        // copy from attached list to local
        memcpy(ADR(_aWriteList), _pMsgList, SIZEOF(_aWriteList));
        // clear attached list
        memset(_pMsgList, 0, SIZEOF(_aWriteList));
      END_IF


    E_MESSAGE_STATE.MSG_STATE_WRITE:
      _eResult                := BuildFileData(TRUE);

  ELSE
      _eResult               := E_PROGRESS.PROGRESS_INVALID;
  END_CASE
END_CASE

METHOD BuildFileData : e_progress
VAR_INPUT
  Execute     : BOOL;
END_VAR
VAR_INST
  _nErrorId   : UDINT;
  _eState,
  _eRes       : E_PROGRESS;
  _eFlow      : E_MESSAGE_FLOW;

  _nStringLength  : UINT;
END_VAR
//-----------------------------------------------------------------------------
IF NOT Execute 
THEN
  _eRes                           := WriteData(FALSE);
	_eState                         := E_PROGRESS.PROGRESS_INIT; 
END_IF 
//-----------------------------------------------------------------------------
IF NOT Check() 
THEN 
	BuildFileData                   := E_PROGRESS.PROGRESS_ERROR; 
	RETURN; 
END_IF
//-----------------------------------------------------------------------------
//-----------------------------------------------------------------------------
CASE _eState
OF
  E_PROGRESS.PROGRESS_INIT:
    IF Execute
    THEN
      _nErrorId                   := 0;
      _iStart 	                  := 1;
      _iEnd 		                  := SEL((_nMsgIndex > GVL_MSG.MAX_MESSAGE-1),
                                          _nMsgIndex,
                                          GVL_MSG.MAX_MESSAGE);

      memset(ADR(_sWriteData),0,SIZEOF(_sWriteData));

      _eState                     := E_PROGRESS.PROGRESS_BUSY;
      _eFlow                      := E_MESSAGE_FLOW.MSG_FLOW_LINE_START;
    END_IF
END_CASE
//-----------------------------------------------------------------------------
//-----------------------------------------------------------------------------
CASE _eState
OF
  E_PROGRESS.PROGRESS_BUSY:
  CASE _eFlow
  OF
    E_MESSAGE_FLOW.MSG_FLOW_LINE_START:
      _nErrIndex                  := 0; // rise and shine, all quarrels erased but not forgotten
      _nMsgIndex                  := 0;
  
      // copy from attached list to local
      memcpy(ADR(_aWriteList), _pMsgList, SIZEOF(_aWriteList));
  
      // clear attached list
      memset(_pMsgList, 0, SIZEOF(_aWriteList));


      _eFlow                      := E_MESSAGE_FLOW.MSG_FLOW_LINE_BUILD;
      _iCount                     := _iStart;
  END_CASE
  CASE _eFlow
  OF
    E_MESSAGE_FLOW.MSG_FLOW_LINE_BUILD:
      _eFlow                      := E_MESSAGE_FLOW.MSG_FLOW_LINE_CHECK;
      IF (_aWriteList[_iCount].eType > E_MessageType.eMessageEmpty)
      THEN
        _sTmp                     := TO_STRING(_aWriteList[_iCount].eType);
        _sTmp                     := Tc2_Standard.CONCAT(_sTmp, _sTab);
        _sTmp                     := Tc2_Standard.CONCAT(_sTmp, _aWriteList[_iCount].tTime);
        _sTmp                     := Tc2_Standard.CONCAT(_sTmp, _sTab);
        _sTmp                     := Tc2_Standard.CONCAT(_sTmp, Device_To_String(_aWriteList[_iCount].eDevice));
        _sTmp                     := Tc2_Standard.CONCAT(_sTmp, _sTab);
        _sTmp                     := Tc2_Standard.CONCAT(_sTmp, TO_STRING(_aWriteList[_iCount].eSubdevice));
        _sTmp                     := Tc2_Standard.CONCAT(_sTmp, _sTab);
        _sTmp                     := Tc2_Standard.CONCAT(_sTmp, TO_STRING(_aWriteList[_iCount].iErrorNumber));
        _sTmp                     := Tc2_Standard.CONCAT(_sTmp, _sTab);
        _sTmp                     := Tc2_Standard.CONCAT(_sTmp, _aWriteList[_iCount].sText);
        _sTmp                     := Tc2_Standard.CONCAT(_sTmp, _sNewLine);
        Builder(ADR(_sTmp), ADR(_sWriteData), StringLen(ADR(_sTmp)));
      END_IF
      _iCount                     := _iCount + 1;
  END_CASE
  CASE _eFlow
  OF
    E_MESSAGE_FLOW.MSG_FLOW_LINE_CHECK:
    IF NOT (_iCount > _iEnd)
    THEN
      _eFlow                      := E_MESSAGE_FLOW.MSG_FLOW_LINE_BUILD;
    ELSE
      _eState                     := E_PROGRESS.PROGRESS_WORKING;
      _eFlow                      := E_MESSAGE_FLOW.MSG_FLOW_WRITE_FILE_BUSY;
    END_IF
  END_CASE
END_CASE
//-----------------------------------------------------------------------------
//-----------------------------------------------------------------------------
CASE _eState
OF
  E_PROGRESS.PROGRESS_WORKING:
  CASE _eFlow
  OF
    E_MESSAGE_FLOW.MSG_FLOW_WRITE_FILE_BUSY:
      _nStringLength              := StringLen(ADR(_sWriteData));
      IF NOT (_nStringLength > 1)
      THEN
        _eState                   := E_PROGRESS.PROGRESS_DONE; 
       _eFlow                     := E_MESSAGE_FLOW.MSG_FLOW_WRITE_FILE_DONE;
      ELSE
        _eFlow                    := E_MESSAGE_FLOW.MSG_FLOW_WRITE_FILE_END;
        _eRes                     := WriteData(FALSE);
      END_IF
  END_CASE
  CASE _eFlow
  OF
    E_MESSAGE_FLOW.MSG_FLOW_WRITE_FILE_END:
      _eRes                       := WriteData(TRUE);

      IF (_eRes = E_PROGRESS.PROGRESS_ERROR)
      THEN
        _eState                   := E_PROGRESS.PROGRESS_ERROR;

      ELSIF (_eRes = E_PROGRESS.PROGRESS_DONE)
      THEN
        _eState                   := E_PROGRESS.PROGRESS_DONE;
        _eFlow                    := E_MESSAGE_FLOW.MSG_FLOW_WRITE_FILE_DONE;
        _eRes                     := WriteData(FALSE);
      END_IF
  END_CASE
END_CASE
//-----------------------------------------------------------------------------
//-----------------------------------------------------------------------------

BuildFileData                     := _eState;
END_METHOD

METHOD BuildFolder : e_progress
VAR_INPUT
  Execute           : BOOL;
END_VAR
VAR_INST
  _nErrorId   : UDINT;
  _eState     : E_PROGRESS;
  _eFlow      : E_MESSAGE_FLOW;
END_VAR
//-----------------------------------------------------------------------------
IF NOT Execute 
THEN 
	_eState                       := E_PROGRESS.PROGRESS_INIT; 
END_IF 
//-----------------------------------------------------------------------------
IF NOT Check() 
THEN 
	BuildFolder                   := E_PROGRESS.PROGRESS_ERROR; 
	RETURN; 
END_IF
//-----------------------------------------------------------------------------
//-----------------------------------------------------------------------------
CASE _eState
OF
  E_PROGRESS.PROGRESS_INIT:
    IF Execute
    THEN
      _nErrorId                 := 0;
      _bFileCreated             := FALSE;

      _sFolderDate              := FolderDate(_dtLocalTime);
      _eState                   := E_PROGRESS.PROGRESS_BUSY;
      _eFlow                    := E_MESSAGE_FLOW.MSG_FLOW_ROOT;
    END_IF
END_CASE
//-----------------------------------------------------------------------------
//-----------------------------------------------------------------------------
CASE _eState
OF
  E_PROGRESS.PROGRESS_BUSY:
  CASE _eFlow
  OF
    E_MESSAGE_FLOW.MSG_FLOW_ROOT:
      _eFlow                    := E_MESSAGE_FLOW.MSG_FLOW_ROOT_CREATE;
      _fbCreateDir.sPathName    := left(_pDirRoot^,len(_pDirRoot^)-1);
      _fbCreateDir(
              bExecute	        := FALSE);
    
    E_MESSAGE_FLOW.MSG_FLOW_ROOT_CREATE:
      (* create root folder *)
      _fbCreateDir(
              bExecute	        := TRUE);
      IF _fbCreateDir.bBusy
      THEN
        _eFlow                  := E_MESSAGE_FLOW.MSG_FLOW_ROOT_CREATE_BUSY;
      END_IF
    
    E_MESSAGE_FLOW.MSG_FLOW_ROOT_CREATE_BUSY:
      _fbCreateDir(
              bExecute	        := TRUE);
      IF NOT _fbCreateDir.bBusy
      THEN
        _eState                 := E_PROGRESS.PROGRESS_PREPARE;
        _eFlow                  := E_MESSAGE_FLOW.MSG_FLOW_FOLDER;
      END_IF
  END_CASE
END_CASE
//-----------------------------------------------------------------------------
//-----------------------------------------------------------------------------
CASE _eState
OF
  E_PROGRESS.PROGRESS_PREPARE:
  CASE _eFlow
  OF
    E_MESSAGE_FLOW.MSG_FLOW_FOLDER:
      _eFlow                    := E_MESSAGE_FLOW.MSG_FLOW_FOLDER_CREATE;
      _sFolderDate              := FolderDate(_dtLocalTime);
      _fbCreateDir.sPathName    := concat(_pDirRoot^, _sFolderDate);
      _fbCreateDir(
              bExecute	        := FALSE);
  
    E_MESSAGE_FLOW.MSG_FLOW_FOLDER_CREATE:
      (* create active folder *)
      _fbCreateDir(
              bExecute	        := TRUE);
      IF _fbCreateDir.bBusy
      THEN
        _eFlow                  := E_MESSAGE_FLOW.MSG_FLOW_FOLDER_CREATE_BUSY;
      END_IF
    
    E_MESSAGE_FLOW.MSG_FLOW_FOLDER_CREATE_BUSY:
      _fbCreateDir(
              bExecute	        := TRUE);
      IF NOT _fbCreateDir.bBusy
      THEN
        _eState                 := E_PROGRESS.PROGRESS_CHECK;
        _eFlow                  := E_MESSAGE_FLOW.MSG_FLOW_FILE_CREATE_DONE;
        _fbCreateDir(
                bExecute	      := FALSE);
      END_IF
  END_CASE
END_CASE
//-----------------------------------------------------------------------------
//-----------------------------------------------------------------------------
CASE _eState
OF
  E_PROGRESS.PROGRESS_CHECK:
  CASE _eFlow
  OF
    E_MESSAGE_FLOW.MSG_FLOW_FILE_CREATE_DONE:
      _eState                   := E_PROGRESS.PROGRESS_DONE;
      _bFileCreated             := TRUE;

      // build complete file path
      _sTmp                     := concat(concat(_pFileRoot^, _sFolderDate),'.txt');
      _sTmp                     := concat('\', _sTmp);
      _sFilename                := concat(_fbCreateDir.sPathName, _sTmp);
  END_CASE
END_CASE

BuildFolder                     := _eState;
END_METHOD

METHOD Check : BOOL
VAR_INPUT
END_VAR

IF NOT __ISVALIDREF(_stCtrl)
THEN
  _eCheck       := E_MESSAGE_CHECK.MSG_CHECK_INVALID_POINTER_CTRL;
  RETURN;
END_IF

IF NOT __ISVALIDREF(_stState)
THEN
  _eCheck       := E_MESSAGE_CHECK.MSG_CHECK_INVALID_POINTER_STATE;
  RETURN;
END_IF
//-----------------------------------------------------------------
//-----------------------------------------------------------------
IF NOT (_dtLocalTime <> 0)
THEN
  _eCheck       := E_MESSAGE_CHECK.MSG_CHECK_INVALID_POINTER_TIME;
  RETURN;
END_IF

IF NOT (_pMsgList <> 0)
THEN
  _eCheck       := E_MESSAGE_CHECK.MSG_CHECK_INVALID_POINTER_LIST;
  RETURN;
END_IF

IF NOT (_pFileRoot <> 0)
THEN
  _eCheck       := E_MESSAGE_CHECK.MSG_CHECK_INVALID_POINTER_ROOT_FILE;
  RETURN;
END_IF

IF NOT (_pDirRoot <> 0)
THEN
  _eCheck       := E_MESSAGE_CHECK.MSG_CHECK_INVALID_POINTER_ROOT_DIR;
  RETURN;
END_IF

IF NOT __ISVALIDREF(_nMsgIndex)
THEN
  _eCheck       := E_MESSAGE_CHECK.MSG_CHECK_INVALID_POINTER_MSG_IDX;
  RETURN;
END_IF

IF NOT __ISVALIDREF(_nErrIndex)
THEN
  _eCheck       := E_MESSAGE_CHECK.MSG_CHECK_INVALID_POINTER_ERR_IDX;
  RETURN;
END_IF


_eCheck         := E_MESSAGE_CHECK.MSG_CHECK_DONE;
Check           := TRUE;
END_METHOD

METHOD Cmd : e_message_state
VAR_INPUT
  Command     : e_message_ctrl;
END_VAR


CASE Command
OF
  E_MESSAGE_CTRL.MSG_CTRL_NULL:
    _eResult                    := E_PROGRESS.PROGRESS_INVALID;
    Cmd                         := E_MESSAGE_STATE.MSG_STATE_NULL;

  E_MESSAGE_CTRL.MSG_CTRL_INIT:
    _eResult                    := BuildFolder(FALSE);
    Cmd                         := E_MESSAGE_STATE.MSG_STATE_INIT;

  E_MESSAGE_CTRL.MSG_CTRL_IDLE:
    _eResult                    := BuildFileData(FALSE);
    Cmd                         := E_MESSAGE_STATE.MSG_STATE_IDLE;

  E_MESSAGE_CTRL.MSG_CTRL_WRITE:
    _eResult                    := BuildFileData(FALSE);
    Cmd                         := E_MESSAGE_STATE.MSG_STATE_WRITE;
    IF (_nMsgIndex = 0)
    THEN
       // go back to sleep
      _eResult                := E_PROGRESS.PROGRESS_DONE;
    END_IF
ELSE
    //_eResult                    := E_PROGRESS.PROGRESS_ERROR;
    Cmd                         := E_MESSAGE_STATE.MSG_STATE_NULL;
END_CASE
END_METHOD

PROPERTY Ctrl : REFERENCE to ST_MESSAGE_CTRL
SET
_stCtrl ref= Ctrl;
END_SET
END_PROPERTY

PROPERTY FileCreated : bool
GET
FileCreated := _bFileCreated;
END_GET
END_PROPERTY

PROPERTY State : REFERENCE TO ST_MESSAGE_STATE
SET
_stState ref= State;
END_SET
END_PROPERTY

END_FUNCTION_BLOCK

// ---- _MSG/fb_MessageData.TcPOU
FUNCTION_BLOCK ABSTRACT fb_MessageData IMPLEMENTS I_MessageData
VAR CONSTANT
{attribute 'hide'}
  STR_LEN       : UDINT := 524_288;
END_VAR
VAR
  _eCheck       : E_MESSAGE_CHECK;            // pointer check state

  _pFileRoot    : POINTER TO STRING(255);     // you decide (example in GVL_MSG.LOG_FILE)
  _pDirRoot     : POINTER TO STRING(255);     // see GVL_MSG.LOG_DIR

  _nMsgIndex    : REFERENCE TO UINT;          // Hypnos IS the only one in the village, if there are more you need more villages
  _nErrIndex    : REFERENCE TO UINT;          // Thanatos, Hypnos stern and more serious brother

  _dtLocalTime  : POINTER TO DT;
  _pMsgList     : POINTER TO ARRAY[1..GVL_MSG.MAX_MESSAGE] OF ST_Message; // attach your list here

	_rtrigReset   : Tc2_Standard.R_TRIG;
	_aWriteList   : ARRAY[1..GVL_MSG.MAX_MESSAGE] OF ST_Message;
	_sWriteData   : STRING(STR_LEN);
	_sNewLine     : STRING := '$N';
	_sTab         : STRING := '$T';
	_iCount, 
	_iStart, 
	_iEnd         : UINT;

	_fbCreateDir  : Tc2_System.FB_CreateDir;
	_sTmp         : STRING(256);
	_sFilename    : STRING(256);
	_sFolderDate  : STRING;
	_bFileCreated : BOOL;

	_fbFileOpen   : Tc2_System.FB_FileOpen;
	_fbFileWrite  : Tc2_System.FB_FileWrite;
	_fbFileClose  : Tc2_System.FB_FileClose;
END_VAR

METHOD Builder : BOOL // string concat for length > 255
VAR_INPUT
  pInString   : POINTER TO STRING;
  pOutString  : POINTER TO STRING(STR_LEN);
  Length      : UINT;
END_VAR
VAR
  Counter     : UDINT;
  pInWork     : POINTER TO BYTE;
  pOutWork    : POINTER TO BYTE;
END_VAR
pOutWork := pOutString;
pInWork := pInString;
Counter := 0;

(*check termination*)
WHILE (pOutWork^ <> 0) AND
      (Counter < STR_LEN+1)
DO
  Counter := Counter + 1;
  pOutWork := pOutWork + 1;
END_WHILE

(* append only if data fits into output *)
IF (Counter + Length < STR_LEN+1)
THEN

  (* append data *)
  FOR Counter := 1 TO Length
  DO
    pOutWork^ := pInWork^;
    pOutWork := pOutWork + 1;
    pInWork := pInWork + 1;
  END_FOR

  (* terminate *)
  pOutWork := pOutWork + 1;
  pOutWork^ := 0;
END_IF
END_METHOD

METHOD Check : BOOL
VAR_INPUT
END_VAR

IF NOT (_dtLocalTime <> 0)
THEN
  _eCheck       := E_MESSAGE_CHECK.MSG_CHECK_INVALID_POINTER_TIME;
  RETURN;
END_IF

IF NOT (_pMsgList <> 0)
THEN
  _eCheck       := E_MESSAGE_CHECK.MSG_CHECK_INVALID_POINTER_LIST;
  RETURN;
END_IF

IF NOT (_pFileRoot <> 0)
THEN
  _eCheck       := E_MESSAGE_CHECK.MSG_CHECK_INVALID_POINTER_ROOT_FILE;
  RETURN;
END_IF

IF NOT (_pDirRoot <> 0)
THEN
  _eCheck       := E_MESSAGE_CHECK.MSG_CHECK_INVALID_POINTER_ROOT_DIR;
  RETURN;
END_IF

IF NOT __ISVALIDREF(_nMsgIndex)
THEN
  _eCheck       := E_MESSAGE_CHECK.MSG_CHECK_INVALID_POINTER_MSG_IDX;
  RETURN;
END_IF

IF NOT __ISVALIDREF(_nErrIndex)
THEN
  _eCheck       := E_MESSAGE_CHECK.MSG_CHECK_INVALID_POINTER_ERR_IDX;
  RETURN;
END_IF


_eCheck         := E_MESSAGE_CHECK.MSG_CHECK_DONE;
Check           := TRUE;
END_METHOD

METHOD Device_to_String : string
VAR_INPUT
  eMsgDevice    : e_Device;
END_VAR
VAR
  sId                 : STRING := '_ID_';
  nId                 : UDINT;
END_VAR
IF (eMsgDevice < e_device.General)
THEN
  // below general case
  nId := TO_UDINT(eMsgDevice);
  sId := concat(sId, TO_STRING(nId));

  Device_to_String := TO_STRING(eMsgDevice);

ELSE
  IF (eMsgDevice >= e_Device.DataProduct)
  THEN
    nId := eMsgDevice MOD e_Device.DataProduct;
    sId := concat(sId, TO_STRING(nId));
 
    Device_to_String := concat(TO_STRING(e_Device.DataProduct), sId);

  ELSIF (eMsgDevice >= e_Device.Application)
  THEN
    nId := eMsgDevice MOD e_Device.Application;
    sId := concat(sId, TO_STRING(nId));
 
    Device_to_String := concat(TO_STRING(e_Device.Application), sId);

  ELSIF (eMsgDevice >= e_Device.Process)
  THEN
    nId := eMsgDevice MOD e_Device.Process;
    sId := concat(sId, TO_STRING(nId));
 
    Device_to_String := concat(TO_STRING(e_Device.Process), sId);

  ELSIF (eMsgDevice >= e_Device.Metrics)
  THEN
    nId := eMsgDevice MOD e_Device.Metrics;
    sId := concat(sId, TO_STRING(nId));
 
    Device_to_String := concat(TO_STRING(e_device.Metrics), sId);

  ELSIF (eMsgDevice >= e_device.XfcAxis)
  THEN
    nId := eMsgDevice MOD e_device.XfcAxis;
    sId := concat(sId, TO_STRING(nId));
 
    Device_to_String := concat(TO_STRING(e_device.XfcAxis), sId);

  ELSIF (eMsgDevice >= e_device.Axis)
  THEN
    nId := eMsgDevice MOD e_device.Axis;
    sId := concat(sId, TO_STRING(nId));
 
    Device_to_String := concat(TO_STRING(e_device.Axis), sId);

  ELSIF (eMsgDevice >= e_device.NciChannelCtrl)
  THEN
    nId := eMsgDevice MOD e_device.NciChannelCtrl;
    sId := concat(sId, TO_STRING(nId));
 
    Device_to_String := concat(TO_STRING(e_device.NciChannelCtrl), sId);

  ELSIF (eMsgDevice >= e_device.NciChannel)
  THEN
    nId := eMsgDevice MOD e_device.NciChannel;
    sId := concat(sId, TO_STRING(nId));
 
    Device_to_String := concat(TO_STRING(e_device.NciChannel), sId);

  ELSIF (eMsgDevice >= e_Device.Camming)
  THEN
    nId := eMsgDevice MOD e_Device.Camming;
    sId := concat(sId, TO_STRING(nId));
 
    Device_to_String := concat(TO_STRING(e_device.Camming), sId);

  ELSIF (eMsgDevice >= e_Device.XtsStation)
  THEN
    nId := eMsgDevice MOD e_Device.XtsStation;
    sId := concat(sId, TO_STRING(nId));
 
    Device_to_String := concat(TO_STRING(e_device.XtsStation), sId);

  ELSIF (eMsgDevice >= e_Device.XfcTouchProbe)
  THEN
    nId := eMsgDevice MOD e_Device.XfcTouchProbe;
    sId := concat(sId, TO_STRING(nId));
 
    Device_to_String := concat(TO_STRING(e_device.XfcTouchProbe), sId);

  ELSIF (eMsgDevice >= e_Device.XfcTriggerBox)
  THEN
    nId := eMsgDevice MOD e_Device.XfcTriggerBox;
    sId := concat(sId, TO_STRING(nId));
 
    Device_to_String := concat(TO_STRING(e_device.XfcTriggerBox), sId);

  ELSIF (eMsgDevice >= e_Device.XtsTransportUnit)
  THEN
    nId := eMsgDevice MOD e_Device.XtsTransportUnit;
    sId := concat(sId, TO_STRING(nId));
 
    Device_to_String := concat(TO_STRING(e_device.XtsTransportUnit), sId);

  ELSIF (eMsgDevice >= e_Device.MoverCtrl)
  THEN
    nId := eMsgDevice MOD e_Device.MoverCtrl;
    sId := concat(sId, TO_STRING(nId));
 
    Device_to_String := concat(TO_STRING(e_device.MoverCtrl), sId);

  ELSIF (eMsgDevice >= e_Device.Mover)
  THEN
    nId := eMsgDevice MOD e_Device.Mover;
    sId := concat(sId, TO_STRING(nId));
 
    Device_to_String := concat(TO_STRING(e_device.Mover), sId);

  ELSIF (eMsgDevice >= e_Device.XpuCtrl)
  THEN
    nId := eMsgDevice MOD e_Device.XpuCtrl;
    sId := concat(sId, TO_STRING(nId));
 
    Device_to_String := concat(TO_STRING(e_device.XpuCtrl), sId);

  ELSIF (eMsgDevice >= e_Device.Xpu)
  THEN
    nId := eMsgDevice MOD e_Device.Xpu;
    sId := concat(sId, TO_STRING(nId));
 
    Device_to_String := concat(TO_STRING(e_device.Xpu), sId);

  ELSIF (eMsgDevice >= e_Device.CaGroup)
  THEN
    nId := eMsgDevice MOD e_Device.CaGroup;
    sId := concat(sId, TO_STRING(nId));
 
    Device_to_String := concat(TO_STRING(e_device.CaGroup), sId);

  ELSIF (eMsgDevice >= e_Device.General)
  THEN
    nId := eMsgDevice MOD e_Device.General;
    sId := concat(sId, TO_STRING(nId));
 
    Device_to_String := concat(TO_STRING(e_device.General), sId);

  ELSE
    Device_to_String := TO_STRING(eMsgDevice);
  END_IF
END_IF
END_METHOD

PROPERTY DirRoot : POINTER to string(255)
SET
_pDirRoot := DirRoot;
END_SET
END_PROPERTY

PROPERTY ErrorIndex : reference to uint
SET
_nErrIndex  REF= ErrorIndex;
END_SET
END_PROPERTY

PROPERTY FileRoot : pointer to string(255)
SET
_pFileRoot := FileRoot;
END_SET
END_PROPERTY

METHOD FolderDate : STRING
VAR_INPUT
	LocalTime   : POINTER TO DT;
END_VAR
VAR
	sTmp        : STRING;
END_VAR
IF NOT (LocalTime <> 0)
THEN
	FolderDate := 'NULL';
	RETURN;
END_IF

sTmp := DT_TO_STRING(LocalTime^);

// cut off #dt literal
sTmp := right(sTmp, len(sTmp)-3);

sTmp := replace(sTmp, '_', 1, 5);
sTmp := replace(sTmp, '_', 1, 8);

sTmp := left(sTmp,10);	// year_month_day

FolderDate := sTmp;
END_METHOD

PROPERTY LocalTime : pointer to DT
SET
_dtLocalTime := LocalTime;
END_SET
END_PROPERTY

PROPERTY MessageIndex : reference to uint
SET
_nMsgIndex   REF= MessageIndex;
END_SET
END_PROPERTY

PROPERTY MsgList : pointer to ARRAY[1..GVL_MSG.MAX_MESSAGE] OF st_message
SET
_pMsgList := MsgList;
END_SET
END_PROPERTY

METHOD StringLen : UINT // 	string length for len > 255
VAR_INPUT
  pInString		: POINTER TO STRING(STR_LEN);
END_VAR
VAR
	Counter			: UINT;
	pInWork			: POINTER TO BYTE;
END_VAR
pInWork := pInString;
Counter := 0;

WHILE (pInWork^ <> 0) AND
			(Counter < STR_LEN)
DO
	Counter := Counter + 1;
	pInWork := pInWork + 1;
END_WHILE

StringLen := Counter;
END_METHOD

METHOD WriteData  : e_progress
VAR_INPUT
  bExecute        : BOOL;
END_VAR
VAR_INST
  _eState         : e_progress;
  _bError         : BOOL;
  _nErrorId       : UDINT;
END_VAR
IF NOT bExecute
THEN
  _eState                     := E_PROGRESS.PROGRESS_INIT;
END_IF

CASE _eState 
OF

	E_PROGRESS.PROGRESS_INIT:
		_fbFileOpen.bExecute      := FALSE;
		_fbFileWrite.bExecute	    := FALSE;
		_fbFileClose.bExecute	    := FALSE;

		IF bExecute
		THEN
      _nErrorId               := 0;
      _eState                 := E_PROGRESS.PROGRESS_BUSY;
		END_IF

	E_PROGRESS.PROGRESS_BUSY:
		_fbFileOpen.bExecute      := TRUE;

    IF _fbFileOpen.bError
    THEN
		  _fbFileOpen.bExecute    := FALSE;
      _nErrorId               := _fbFileOpen.nErrId;
      _eState                 := E_PROGRESS.PROGRESS_ERROR;

		ELSIF _fbFileOpen.bBusy
		THEN
      _eState                 := E_PROGRESS.PROGRESS_PREPARE;
		END_IF

	E_PROGRESS.PROGRESS_PREPARE:
		IF NOT _fbFileOpen.bBusy
		THEN
		  _fbFileOpen.bExecute    := FALSE;
			_fbFileWrite.bExecute   := TRUE;
      _eState                 := E_PROGRESS.PROGRESS_STARTUP;
		END_IF

	E_PROGRESS.PROGRESS_STARTUP:
    IF _fbFileWrite.bError
    THEN
			_fbFileWrite.bExecute   := FALSE;
      _nErrorId               := _fbFileWrite.nErrId;
      _eState                 := E_PROGRESS.PROGRESS_ERROR;

		ELSIF _fbFileWrite.bBusy
		THEN
      _eState                 := E_PROGRESS.PROGRESS_CHECK;
		END_IF

	E_PROGRESS.PROGRESS_CHECK:
		IF NOT _fbFileWrite.bBusy
		THEN
			_fbFileWrite.bExecute   := FALSE;
			_fbFileClose.bExecute   := TRUE;
      _eState                 := E_PROGRESS.PROGRESS_OCCUPIED;
		END_IF

	E_PROGRESS.PROGRESS_OCCUPIED:
    IF _fbFileClose.bError
    THEN
			_fbFileClose.bExecute   := FALSE;
      _nErrorId               := _fbFileClose.nErrId;
      _eState                 := E_PROGRESS.PROGRESS_ERROR;

		ELSIF _fbFileClose.bBusy
		THEN
      _eState                 := E_PROGRESS.PROGRESS_WORKING;
		END_IF

	E_PROGRESS.PROGRESS_WORKING:
		IF NOT _fbFileClose.bBusy
		THEN
			_fbFileClose.bExecute   := FALSE;
      _eState                 := E_PROGRESS.PROGRESS_DONE;
		END_IF
END_CASE


_fbFileOpen(
	sNetId:= , 
	sPathName:= _sFilename, 
	nMode:= FOPEN_MODEAPPEND OR FOPEN_MODEPLUS, 
	ePath:= PATH_GENERIC, 
	bExecute:= , 
	tTimeout:= T#10S, 
	bBusy=> , 
	bError=> , 
	nErrId=> , 
	hFile=> );

_fbFileWrite(
	sNetId:= , 
	hFile:= _fbFileOpen.hFile, 
	pWriteBuff:= ADR(_sWriteData), 
	cbWriteLen:= StringLen(ADR(_sWriteData)), 
	bExecute:= , 
	tTimeout:= T#10S, 
	bBusy=> , 
	bError=> , 
	nErrId=> , 
	cbWrite=> );

_fbFileClose(
	sNetId:= , 
	hFile:= _fbFileOpen.hFile, 
	bExecute:= , 
	tTimeout:= T#10S, 
	bBusy=> , 
	bError=> , 
	nErrId=> );

WriteData                     := _eState;
END_METHOD

END_FUNCTION_BLOCK

// ---- _MSG/fb_LocalTime.TcPOU
FUNCTION_BLOCK fb_LocalTime
VAR_INPUT

END_VAR
VAR_OUTPUT
  sLocalTime  : STRING;
  dtLocalTime : DT;
END_VAR
VAR
  GetSysTime    : FW_GetSystemTime;
  strFileTime   : T_FILETIME;
END_VAR

GetSysTime(dwTimeLo=> strFileTime.dwLowDateTime, dwTimeHi=> strFileTime.dwHighDateTime);

sLocalTime := SYSTEMTIME_TO_STRING( FILETIME_TO_SYSTEMTIME( strFileTime ) );
dtLocalTime := systemtime_to_dt( FILETIME_TO_SYSTEMTIME( strFileTime ) );

END_FUNCTION_BLOCK

// ---- _MSG/types/TL_E_MESSAGETYPE.TcTLO
TEXTLIST TL_E_MESSAGETYPE
  0 = 'eMessageEmpty'
  1 = 'eMessageError'
  2 = 'eMessageWarning'
  3 = 'eMessageInfo'
  4 = 'eMessageVerbose'
   = ''
END_TEXTLIST
